// TIA Portal V19 export
FUNCTION_BLOCK "SmartLoopControl"   // FB182, LAD
TITLE = SMART LOOP CONTROLLER
// stored: Access Published, MemoryReserve 100, SetENOAutomatically false
   VAR_INPUT
      AreaInterfaceEntry : "AreaInterface";
      AreaInterfaceExit : "AreaInterface";
      DataIn : Struct
         Pb_StartStop : Bool;
         Pb_Start : Bool;
         Pb_Stop : Bool;
         SensorEntryMaterialPresence : Bool;
         SensorExitMaterialPresence : Bool;
         SensorExitEnableUseEncoder : Bool;
         SensorNotLoopMinHigh : Bool;   // FALSE = Min High
         SensorLoopMaxLow_Or_TPEntry : Bool;
         SensorLoopMaxLow_Or_TPExit : Bool;
         PlugConnected : Bool;
      END_STRUCT;
      CIn : "SmartLoopControl_CIn";
      Config : Struct
         PitTables_Exist : Bool := FALSE;
         Entry_PercentagePosError : LReal := 10.0;   // % Max Delta Counter position Vs Positions calculated from velocity
         Exit_PercentagePosError : LReal := 10.0;   // % Max Delta Counter position Vs Positions calculated from velocity
         Delay_CheckNoEntryBkwEnable : Time := T#6s;
         Delay_CheckNoEntryFwdEnable : Time := T#6s;
         Delay_CheckNoExitBkwEnable : Time := T#6s;
         Delay_CheckNoExitFwdEnable : Time := T#6s;
      END_STRUCT;
   END_VAR
   VAR_OUTPUT
      MachineInterfaceEntry : "MachineInterface";
      MachineInterfaceExit : "MachineInterface";
      COut : "SmartLoopControl_COut";
      DataOut : Struct
         LampSystemOn : Bool;
      END_STRUCT;
   END_VAR
   VAR_IN_OUT
      PersistentValues : Struct
         Par : "SmartLoopControl_Par";
      END_STRUCT;
   END_VAR
   VAR
      Ctrl : Struct
         RstAlarms : Bool;
         StopInPhase : Bool;
         StopProgrammed : Bool;
         StopAborting : Bool;
         ForceSyncFirstStart : Bool;
         ForceSyncMinHigh : Bool;
         ForceSyncCyclic : Bool;
         ForceSyncExt : Bool;
         ForceSync : Bool;
         Sync_Exe : Bool;
         Sync_EntryReduceOrStopFeed : Bool;
         Sync_ExitReduceOrStopFeed : Bool;
         MeasuringEnable : Bool;
         Entry_EnableFeedBkw : Bool;
         Entry_EnableFeedFwd : Bool;
         Exit_EnableFeedBkw : Bool;
         Exit_EnableFeedFwd : Bool;
         Entry_VelocityOverride : LReal;
         Exit_VelocityOverride : LReal;
         Exit_MaxAllowableFeedFwd : LReal;
      END_STRUCT;
      Sts : Struct
         IsStandstill : Bool;
         AlarmsPresence : Bool;
         WarningsPresence : Bool;
         SensorsMaxLow_OFF : Bool;
         SensorsMaxLow_ON : Bool;
         LoopMaterialCounterValid : Bool;
         SynchroRunning : Bool;
         CheckSensorCatchIsOn : Bool;
         CheckSensorLooseIsOn : Bool;
         WorkModeMatCounter : Bool;
         WorkModeSensors : Bool;
         SystemOn : Bool;
         MinHighReached : Bool;
         SynchroDone : Bool;
         CntFeedIncValid : Bool;
         AntiRepetitionForceSyncExt : Bool;
         Entry_MeasuringValuePosAxValid : Bool;
         Exit_MeasuringValuePosAxValid : Bool;
         Entry_MeasuringValueMatCounterValid : Bool;
         Exit_MeasuringValueMatCounterValid : Bool;
         SynchroDoneTof2s : Bool;
         MaxLowReached : Bool;
         SelectedPosStopMaxLow : LReal;
         SelectedOverrideScaling : LReal;
         LoopMaterialCounter : LReal;
         DifferenceInc : LReal;
         CntFeedIncPrevious : LReal;
         MissingToCyclicSync : LReal;
         SyncroMemLoopMaterialCounter : LReal;
         AntiRepetitionForceSyncExtSaveEntryMatCounter : LReal;
         AntiRepetitionForceSyncExtSaveExitMatCounter : LReal;
         EncEntry_MeasuringValuePosAx : LReal;
         EncExit_MeasuringValuePosAx : LReal;
         EncEntry_MeasuringValueMatCounter : LReal;
         EncExit_MeasuringValueMatCounter : LReal;
         LoopMaterialCounterOffset : LReal;
         LoopMaterialMissingToMaxLow : LReal;
         LoopMaterialMissingToMinHigh : LReal;
         Cases_Entry_VelocityOverride : UInt;
         Cases_Exit_VelocityOverride : UInt;
         Cases_Exit_MaxFeed : UInt;
         WorkMode : UInt;
      END_STRUCT;
      Wng : Struct
         NoAutReady : Bool;
         MeasInputsXORMeasuringValue : Bool;
         TimeOutCalculateLoopCounterOffset : Bool;
         SensorEnableEncIsOff : Bool;
         Entry_MatCounterNotValid : Bool;
         Exit_MatCounterNotValid : Bool;
         NotSystemOn : Bool;
         MinHighReached : Bool;
         SyncNeedToLooseSensor : Bool;
         SyncNeedToCatchSensor : Bool;
         Entry_NoBkwEnable : Bool;
         Entry_NoFwdEnable : Bool;
         Exit_NoBkwEnable : Bool;
         Exit_NoFwdEnable : Bool;
      END_STRUCT;
      Alr : Struct
         MeasInputsXORInputState : Bool;
         Entry_MatCounterLooseOfValidState : Bool;
         Exit_MatCounterLooseOfValidState : Bool;
         SensorError : Bool;
         PlugNotConnected : Bool;
         SyncSensorNotCatch : Bool;
         SyncSensorNotLoose : Bool;
         Entry_NoCounterMove : Bool;
         Exit_NoCounterMove : Bool;
      END_STRUCT;
      tonCheckMeasInputStateXOR : TON_TIME;
      tonDelaySensorMaxLowLoose { S7_SetPoint := 'True'} : TON_TIME;
      tonDelaySensorMaxLowCatch { S7_SetPoint := 'True'} : TON_TIME;
      tonCheckNoEntryCounterMove { S7_SetPoint := 'True'} : TON_TIME;
      tonCheckNoExitCounterMove { S7_SetPoint := 'True'} : TON_TIME;
      tonEnableForceSyncCyclic { S7_SetPoint := 'True'} : TON_TIME;
      tonSynchIdle { S7_SetPoint := 'True'} : TON_TIME;
      tonCheckBothMeasuringDone { S7_SetPoint := 'True'} : TON_TIME;
      tonTimeOutCalculateCounterOffset { S7_SetPoint := 'True'} : TON_TIME;
      tonSynchAutoReset { S7_SetPoint := 'True'} : TON_TIME;
      tof2sSynchroDone { S7_SetPoint := 'True'} : TON_TIME;
      tonRstMaterialCounterValid { S7_SetPoint := 'True'} : TON_TIME;
      tonSetMaxLow { S7_SetPoint := 'True'} : TON_TIME;
      tonRstMaxLow { S7_SetPoint := 'True'} : TON_TIME;
      tonCheckNoEntryBkwEnable { S7_SetPoint := 'True'} : TON_TIME;
      tonCheckNoEntryFwdEnable { S7_SetPoint := 'True'} : TON_TIME;
      tonCheckNoExitBkwEnable { S7_SetPoint := 'True'} : TON_TIME;
      tonCheckNoExitFwdEnable { S7_SetPoint := 'True'} : TON_TIME;
      SynchCycle { S7_SetPoint := 'True'} : UInt;
      CheckSensorCatchSaveLoopMaterialCounter : LReal;
      CheckSensorCatchFeeding : LReal;
      CheckSensorLooseSaveLoopMaterialCounter : LReal;
      CheckSensorLooseFeeding : LReal;
      AuxPbStartStopOneShot { S7_SetPoint := 'True'} : Bool;
      AuxSyncFirstStartOneShot : Bool;
      ModeMatCounterAndSystemOn : Bool;
      MinHighCumulative : Bool;
      AuxSyncMinHighOneShot : Bool;
      Entry_SaveMesInpID : UInt;
      Exit_SaveMesInpID : UInt;
      Check_Entry_Velocity { S7_SetPoint := 'True'} : "Check_Axis_Velocity";
      Check_Exit_Velocity { S7_SetPoint := 'True'} : "Check_Axis_Velocity";
   END_VAR
   VAR_TEMP
      PosMax : LReal;
      MaxMaterialInsideLoop : LReal;
      DeltaPosSync : LReal;
      DeltaPos : LReal;
      PbStartOneShot : Bool;
      PbStopOneShot : Bool;
      OK : Bool;
      Req : Bool;
      MinHighOverride : Bool;
      RstSynchro : Bool;
   END_VAR
   VAR CONSTANT
      DELTA_POS_LOOP_OVER_LOW_TABLE : LReal := 100.0;
      SYNCH_00_INIT : UInt := 0;
      SYNCH_01_ACTIVATE_MEASINPUTS : UInt := 1;
      SYNCH_10_IDLE : UInt := 10;
      SYNCH_11_CATCH_SENSOR : UInt := 11;
      SYNCH_12_LOOSE_SENSOR : UInt := 12;
      SYNCH_13_LAST_CATCH_SENSOR : UInt := 13;
      SYNCH_14_CALCULATE_COUNTER_OFFSET : UInt := 14;
      SYNCH_90_ERROR : UInt := 90;
      MODE_00_USE_SENSOR : UInt := 0;
      MODE_01_USE_MATERIAL_COUNTERS : UInt := 1;
      ENTRY_CASE_01_V0_ALARM_PRESENCE : UInt := 1;
      ENTRY_CASE_02_V0_MAX_LOW : UInt := 2;
      ENTRY_CASE_03_VMin_MAX_LOW_OVERRIDE : UInt := 3;
      ENTRY_CASE_04_V100_SYSTEM_OFF : UInt := 4;
      ENTRY_CASE_11_VMin_MODE_SENSORS : UInt := 11;
      ENTRY_CASE_12_VMax_MODE_SENSORS : UInt := 12;
      ENTRY_CASE_13_V100_MODE_SENSORS : UInt := 13;
      ENTRY_CASE_21_V100_SYNCHRO_RUNNING : UInt := 21;
      ENTRY_CASE_22_V0_SYNCHRO_RUNNING : UInt := 22;
      ENTRY_CASE_23_VMin_SYNCHRO_RUNNING : UInt := 23;
      ENTRY_CASE_24_VMin_MODE_COUNTERS : UInt := 24;
      ENTRY_CASE_25_VMed_MODE_COUNTERS : UInt := 25;
      ENTRY_CASE_26_VMax_MODE_COUNTERS : UInt := 26;
      ENTRY_CASE_27_VMaxMax_MODE_COUNTERS : UInt := 27;
      ENTRY_CASE_30_V100_UNKNOW : UInt := 30;
      EXIT_CASE_01_V0_ALARM_PRESENCE : UInt := 1;
      EXIT_CASE_02_0_MIN_HIGH : UInt := 2;
      EXIT_CASE_03_VMin_SYSTEM_OFF : UInt := 3;
      EXIT_CASE_04_VMin_NEXT_EMPTYING : UInt := 4;
      EXIT_CASE_05_VMax_EMPTYING : UInt := 5;
      EXIT_CASE_11_V100_MODE_SENSORS_OR_EXIT_MAN : UInt := 11;
      EXIT_CASE_12_VMIN_MODE_SENSORS_TEMPORARY : UInt := 12;
      EXIT_CASE_20_100_SYNCRO_RUNNING : UInt := 20;
      EXIT_CASE_21_0_SYNCRO_RUNNING : UInt := 21;
      EXIT_CASE_22_VMin_SYNCRO_RUNNING : UInt := 22;
      EXIT_CASE_23_VMin_MODE_COUNTERS : UInt := 23;
      EXIT_CASE_24_VMed_MODE_COUNTERS : UInt := 24;
      EXIT_CASE_25_VMax_MODE_COUNTERS : UInt := 25;
      EXIT_CASE_26_100_MODE_COUNTERS : UInt := 26;
      EXIT_MAX_FEED_CASE_1_NO_LIMIT : UInt := 1;
      EXIT_MAX_FEED_CASE_2_SYSTEM_OFF : UInt := 2;
      EXIT_MAX_FEED_CASE_3_NEXT_END_OF_MATERIAL : UInt := 3;
      EXIT_MAX_FEED_CASE_4_LOOP_MAT_COUNTER_NOT_VALID : UInt := 4;
      EXIT_MAX_FEED_CASE_5_LOOP_MAT_COUNTER_VALID : UInt := 5;
      EXIT_MAX_FEED_CASE_6_ALARM : UInt := 6;
      EXIT_MAX_FEED_CASE_7_MIN_HIGH_REACHED : UInt := 7;
   END_VAR
   VAR_TEMP   // added for the SCL form of the ladder/FBD networks
      _w1 : Bool;
      _w2 : Bool;
      _w3 : Bool;
      _w4 : Bool;
   END_VAR
BEGIN

REGION Network 1: Reset alarms
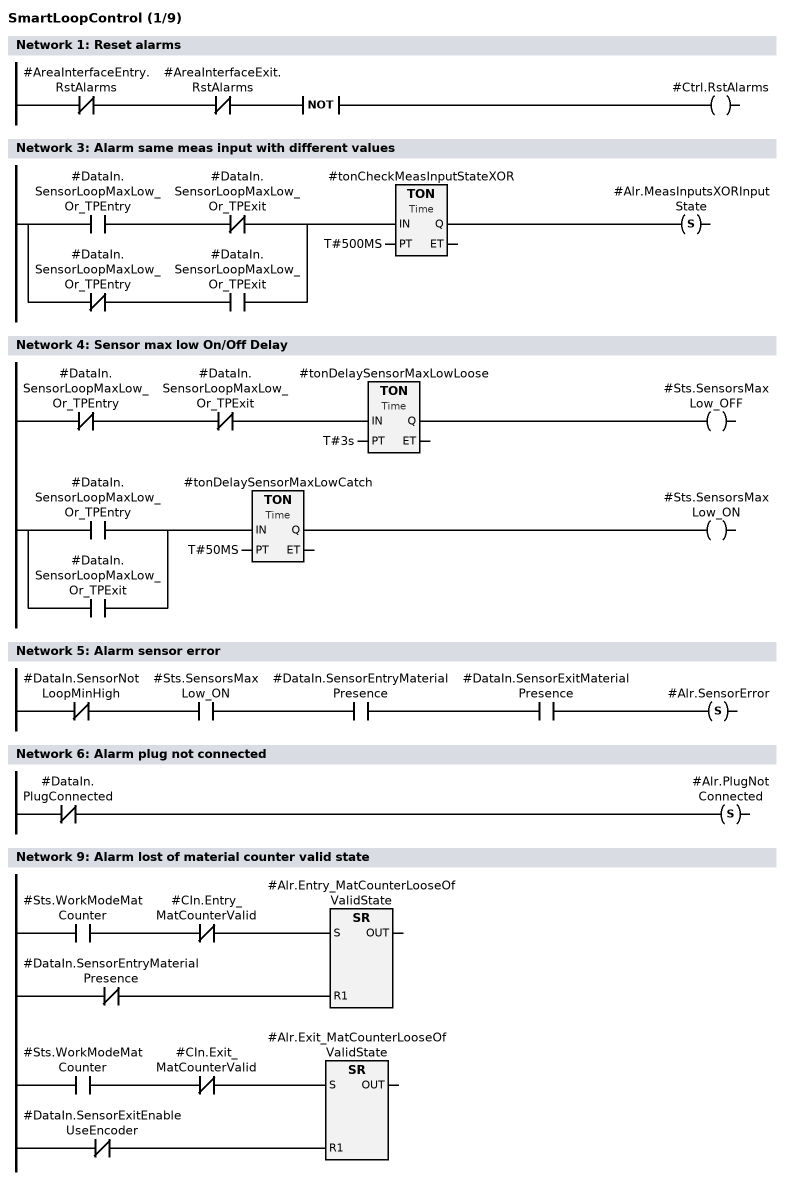
   RUNG wire#powerrail
      I_Contact( #AreaInterfaceEntry.RstAlarms )
      I_Contact( #AreaInterfaceExit.RstAlarms )
      Not()
      Coil( #Ctrl.RstAlarms )
   END_RUNG
   // the same network as SCL:
   #Ctrl.RstAlarms := NOT (NOT #AreaInterfaceEntry.RstAlarms AND NOT #AreaInterfaceExit.RstAlarms);
END_REGION

REGION Network 2 (SCL): Reset alarms execution
   IF #Ctrl.RstAlarms THEN
       #Wng.NoAutReady := FALSE;
       #Wng.MeasInputsXORMeasuringValue := FALSE;
       #Wng.TimeOutCalculateLoopCounterOffset := FALSE;
       #Wng.SensorEnableEncIsOff := FALSE;
       #Wng.Entry_MatCounterNotValid := FALSE;
       #Wng.Exit_MatCounterNotValid := FALSE;
       #Wng.NotSystemOn := FALSE;
       #Wng.MinHighReached := FALSE;
       #Wng.SyncNeedToLooseSensor := FALSE;
       #Wng.SyncNeedToCatchSensor := FALSE;
       #Wng.Entry_NoBkwEnable := FALSE;
       #Wng.Entry_NoFwdEnable := FALSE;
       #Wng.Exit_NoBkwEnable := FALSE;
       #Wng.Exit_NoFwdEnable := FALSE;

       #Alr.MeasInputsXORInputState := FALSE;
       #Alr.Entry_MatCounterLooseOfValidState := FALSE;
       #Alr.Exit_MatCounterLooseOfValidState := FALSE;
       #Alr.SensorError := FALSE;
       #Alr.SyncSensorNotCatch := FALSE;
       #Alr.SyncSensorNotLoose := FALSE;
       #Alr.Entry_NoCounterMove := FALSE;
       #Alr.Exit_NoCounterMove := FALSE;
       #Alr.PlugNotConnected := FALSE;

   END_IF;
END_REGION

REGION Network 3: Alarm same meas input with different values
   RUNG wire#powerrail
      Contact( #DataIn.SensorLoopMaxLow_Or_TPEntry )
      I_Contact( #DataIn.SensorLoopMaxLow_Or_TPExit )
      wire#w1
      { S7_Templates := "time_type := Time" } #tonCheckMeasInputStateXOR.TON(pt := T#500MS, et =>)
      S_Coil( #Alr.MeasInputsXORInputState )
   END_RUNG
   RUNG wire#powerrail
      I_Contact( #DataIn.SensorLoopMaxLow_Or_TPEntry )
      Contact( #DataIn.SensorLoopMaxLow_Or_TPExit )
   END_RUNG wire#w1
   // the same network as SCL:
   #tonCheckMeasInputStateXOR(IN := (#DataIn.SensorLoopMaxLow_Or_TPEntry AND NOT #DataIn.SensorLoopMaxLow_Or_TPExit) OR (NOT #DataIn.SensorLoopMaxLow_Or_TPEntry AND #DataIn.SensorLoopMaxLow_Or_TPExit),   // TON
                           PT := T#500MS);
   IF #tonCheckMeasInputStateXOR.Q THEN #Alr.MeasInputsXORInputState := TRUE; END_IF;
END_REGION

REGION Network 4: Sensor max low On/Off Delay
   RUNG wire#powerrail
      I_Contact( #DataIn.SensorLoopMaxLow_Or_TPEntry )
      I_Contact( #DataIn.SensorLoopMaxLow_Or_TPExit )
      { S7_Templates := "time_type := Time" } #tonDelaySensorMaxLowLoose.TON(pt := T#3s, et =>)
      Coil( #Sts.SensorsMaxLow_OFF )
   END_RUNG
   RUNG wire#powerrail
      Contact( #DataIn.SensorLoopMaxLow_Or_TPEntry )
      wire#w1
      { S7_Templates := "time_type := Time" } #tonDelaySensorMaxLowCatch.TON(pt := T#50MS, et =>)
      Coil( #Sts.SensorsMaxLow_ON )
   END_RUNG
   RUNG wire#powerrail
      Contact( #DataIn.SensorLoopMaxLow_Or_TPExit )
   END_RUNG wire#w1
   // the same network as SCL:
   #tonDelaySensorMaxLowLoose(IN := NOT #DataIn.SensorLoopMaxLow_Or_TPEntry AND NOT #DataIn.SensorLoopMaxLow_Or_TPExit,   // TON
                           PT := T#3s);
   #Sts.SensorsMaxLow_OFF := #tonDelaySensorMaxLowLoose.Q;
   #tonDelaySensorMaxLowCatch(IN := #DataIn.SensorLoopMaxLow_Or_TPEntry OR #DataIn.SensorLoopMaxLow_Or_TPExit,   // TON
                           PT := T#50MS);
   #Sts.SensorsMaxLow_ON := #tonDelaySensorMaxLowCatch.Q;
END_REGION

REGION Network 5: Alarm sensor error
   RUNG wire#powerrail
      I_Contact( #DataIn.SensorNotLoopMinHigh )
      Contact( #Sts.SensorsMaxLow_ON )
      Contact( #DataIn.SensorEntryMaterialPresence )
      Contact( #DataIn.SensorExitMaterialPresence )
      S_Coil( #Alr.SensorError )
   END_RUNG
   // the same network as SCL:
   IF NOT #DataIn.SensorNotLoopMinHigh AND #Sts.SensorsMaxLow_ON AND #DataIn.SensorEntryMaterialPresence AND #DataIn.SensorExitMaterialPresence THEN
       #Alr.SensorError := TRUE;
   END_IF;
END_REGION

REGION Network 6: Alarm plug not connected
   RUNG wire#powerrail
      I_Contact( #DataIn.PlugConnected )
      S_Coil( #Alr.PlugNotConnected )
   END_RUNG
   // the same network as SCL:
   IF NOT #DataIn.PlugConnected THEN #Alr.PlugNotConnected := TRUE; END_IF;
END_REGION

REGION Network 7 (SCL): Switch position Max Low / Middle as used Max Low
   IF  NOT #CIn.MaterialMiddlePos_Request
   THEN
       #Sts.SelectedPosStopMaxLow := #PersistentValues.Par.PosStopMaxLow;
       #Sts.SelectedOverrideScaling := 1.0;

   ELSE
       // Force value of middle position if is not properly setting
       IF NOT (#PersistentValues.Par.PosStopMiddle > #PersistentValues.Par.PosStopMinHigh
           AND
           #PersistentValues.Par.PosStopMiddle < #PersistentValues.Par.PosStopMaxLow)
       THEN
           #PersistentValues.Par.PosStopMiddle := #PersistentValues.Par.PosStopMinHigh + ((#PersistentValues.Par.PosStopMaxLow - #PersistentValues.Par.PosStopMinHigh) / 2.0);
       END_IF;

       // the new position for max low is the middle pistion
       #Sts.SelectedPosStopMaxLow := #PersistentValues.Par.PosStopMiddle;

       // this ratio is apply to all the position refered to max low (e.g. the limits for change exit velocity override)
       #Sts.SelectedOverrideScaling := #PersistentValues.Par.PosStopMiddle / #PersistentValues.Par.PosStopMaxLow;






   END_IF;
END_REGION

REGION Network 8 (SCL): Alarms Synch sensor (table) NOT catch / loose
   // !!! Se per qualche motivo il sensore di ansa bassa rimane sempre ON o sempre OFF c'è il rischio che durante il sincronismo dell'ansa no si verifichi mai l'evento di "sensore catturato" o "sensore perso" con conseguente riempimento eccessivo della
   // lamiera in ansa..Questi allami allarmi verificano se la quantità di lamiera rispetto al momento in cui è iniziato il controllo ha un valore coerente con la massima quantità possibile.
   #PosMax := MAX_LREAL(IN1 := #Sts.SelectedPosStopMaxLow, IN2 := #PersistentValues.Par.PosSynch);
   #MaxMaterialInsideLoop := #PosMax - #PersistentValues.Par.PosStopMinHigh;


   IF #Sts.LoopMaterialCounterValid AND #Sts.SynchroRunning THEN
       IF ((#SynchCycle = #SYNCH_11_CATCH_SENSOR) OR (#SynchCycle = #SYNCH_13_LAST_CATCH_SENSOR))
           AND NOT #Alr.SyncSensorNotCatch AND NOT #Sts.CheckSensorCatchIsOn
       THEN
           #Sts.CheckSensorCatchIsOn := TRUE;
           #CheckSensorCatchSaveLoopMaterialCounter := #Sts.LoopMaterialCounter;
       ELSIF ((#SynchCycle = #SYNCH_11_CATCH_SENSOR) OR (#SynchCycle = #SYNCH_13_LAST_CATCH_SENSOR))
           AND NOT #Alr.SyncSensorNotCatch AND #Sts.CheckSensorCatchIsOn
       THEN
           #CheckSensorCatchFeeding := ABS(#Sts.LoopMaterialCounter - #CheckSensorCatchSaveLoopMaterialCounter);
           IF #CheckSensorCatchFeeding > (1.5 * #MaxMaterialInsideLoop) THEN
               #Alr.SyncSensorNotCatch := TRUE;
           END_IF;
       ELSE
           #Sts.CheckSensorCatchIsOn := FALSE;
       END_IF;

       IF #SynchCycle = #SYNCH_12_LOOSE_SENSOR AND
           NOT #Alr.SyncSensorNotLoose AND NOT #Sts.CheckSensorLooseIsOn
       THEN
           #Sts.CheckSensorLooseIsOn := TRUE;
           #CheckSensorLooseSaveLoopMaterialCounter := #Sts.LoopMaterialCounter;
       ELSIF #SynchCycle = #SYNCH_12_LOOSE_SENSOR
           AND NOT #Alr.SyncSensorNotLoose AND #Sts.CheckSensorLooseIsOn
       THEN
           #CheckSensorLooseFeeding := ABS(#Sts.LoopMaterialCounter - #CheckSensorLooseSaveLoopMaterialCounter);
           IF #CheckSensorLooseFeeding > (1.5 * #MaxMaterialInsideLoop)
           THEN
               #Alr.SyncSensorNotLoose := TRUE;
           END_IF;
       ELSE
           #Sts.CheckSensorLooseIsOn := FALSE;
       END_IF;
   ELSE
       #Sts.CheckSensorCatchIsOn := FALSE;
       #Sts.CheckSensorLooseIsOn := FALSE;
   END_IF;
END_REGION

REGION Network 9: Alarm lost of material counter valid state
   RUNG wire#powerrail
      Contact( #Sts.WorkModeMatCounter )
      I_Contact( #CIn.Entry_MatCounterValid )
      S_SR(operand := #Alr.Entry_MatCounterLooseOfValidState, r1 := wire#w1)
   END_RUNG
   RUNG wire#powerrail
      I_Contact( #DataIn.SensorEntryMaterialPresence )
   END_RUNG wire#w1
   RUNG wire#powerrail
      Contact( #Sts.WorkModeMatCounter )
      I_Contact( #CIn.Exit_MatCounterValid )
      S_SR(operand := #Alr.Exit_MatCounterLooseOfValidState, r1 := wire#w2)
   END_RUNG
   RUNG wire#powerrail
      I_Contact( #DataIn.SensorExitEnableUseEncoder )
   END_RUNG wire#w2
   // the same network as SCL:
   IF #Sts.WorkModeMatCounter AND NOT #CIn.Entry_MatCounterValid THEN
       #Alr.Entry_MatCounterLooseOfValidState := TRUE;   // SR flip-flop
   END_IF;
   IF NOT #DataIn.SensorEntryMaterialPresence THEN #Alr.Entry_MatCounterLooseOfValidState := FALSE; END_IF;
   IF #Sts.WorkModeMatCounter AND NOT #CIn.Exit_MatCounterValid THEN
       #Alr.Exit_MatCounterLooseOfValidState := TRUE;   // SR flip-flop
   END_IF;
   IF NOT #DataIn.SensorExitEnableUseEncoder THEN #Alr.Exit_MatCounterLooseOfValidState := FALSE; END_IF;
END_REGION

REGION Network 10: Alarm no Entry counter move
   // sys.bypass = cambiare #Config.Entry_PercentagePosError in un 0/1 oppure valore time per il timer #tonCheckNoEntryCounterMove
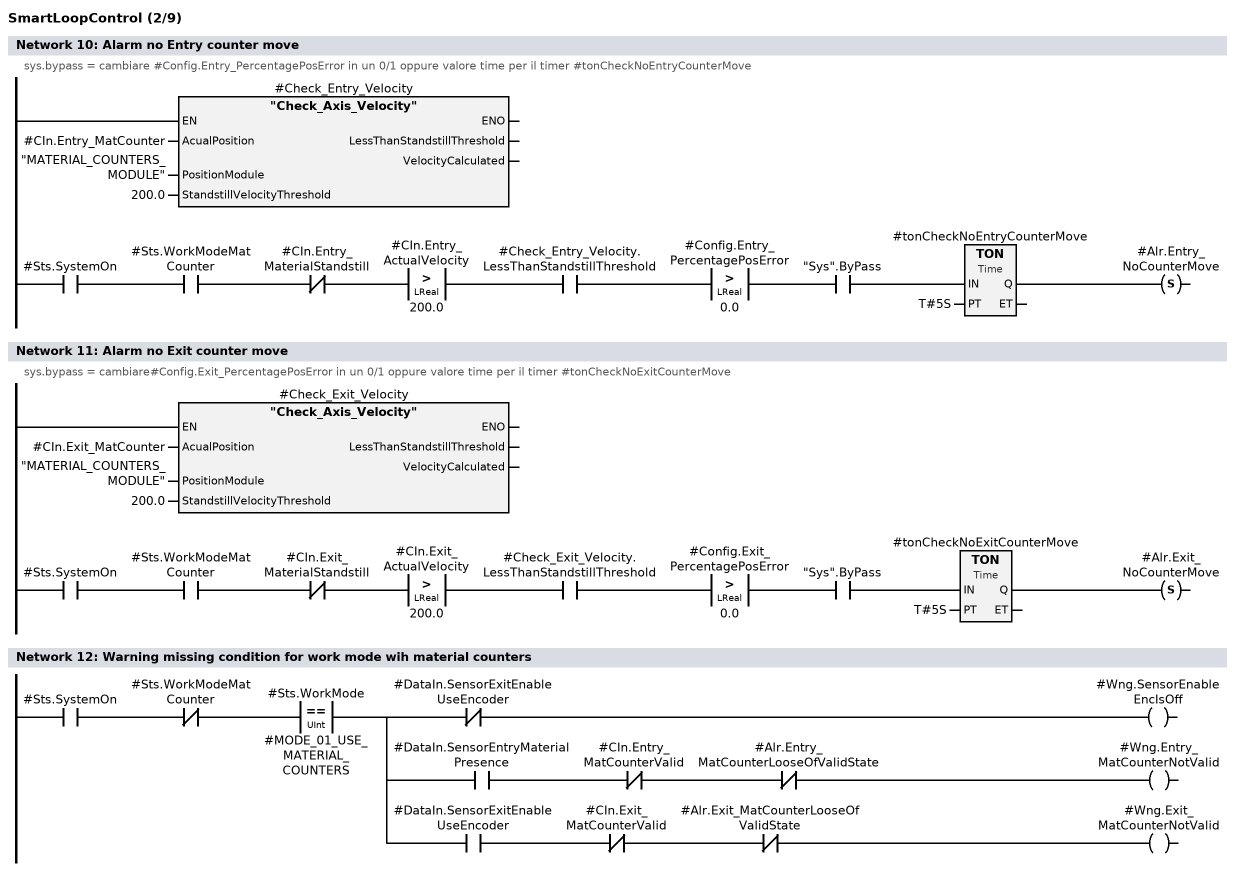
   RUNG wire#powerrail
      #Check_Entry_Velocity(AcualPosition := #CIn.Entry_MatCounter, PositionModule := "MATERIAL_COUNTERS_MODULE", StandstillVelocityThreshold := 200.0, LessThanStandstillThreshold =>, VelocityCalculated =>)
   END_RUNG
   RUNG wire#powerrail
      Contact( #Sts.SystemOn )
      Contact( #Sts.WorkModeMatCounter )
      I_Contact( #CIn.Entry_MaterialStandstill )
      { S7_Templates := "SrcType := LReal" } GT_Contact(in1 := #CIn.Entry_ActualVelocity, in2 := 200.0)
      Contact( #Check_Entry_Velocity.LessThanStandstillThreshold )
      { S7_Templates := "SrcType := LReal" } GT_Contact(in1 := #Config.Entry_PercentagePosError, in2 := 0.0)
      Contact( "Sys".ByPass )
      { S7_Templates := "time_type := Time" } #tonCheckNoEntryCounterMove.TON(pt := T#5S, et =>)
      S_Coil( #Alr.Entry_NoCounterMove )
   END_RUNG
   // the same network as SCL:
   #Check_Entry_Velocity(AcualPosition := #CIn.Entry_MatCounter,   // "Check_Axis_Velocity"
                         PositionModule := "MATERIAL_COUNTERS_MODULE",
                         StandstillVelocityThreshold := 200.0);
   #tonCheckNoEntryCounterMove(IN := #Sts.SystemOn AND #Sts.WorkModeMatCounter AND NOT #CIn.Entry_MaterialStandstill AND (#CIn.Entry_ActualVelocity > 200.0) AND #Check_Entry_Velocity.LessThanStandstillThreshold AND (#Config.Entry_PercentagePosError > 0.0) AND "Sys".ByPass,   // TON
                           PT := T#5S);
   IF #tonCheckNoEntryCounterMove.Q THEN #Alr.Entry_NoCounterMove := TRUE; END_IF;
END_REGION

REGION Network 11: Alarm no Exit counter move
   // sys.bypass = cambiare#Config.Exit_PercentagePosError in un 0/1 oppure valore time per il timer #tonCheckNoExitCounterMove
   RUNG wire#powerrail
      #Check_Exit_Velocity(AcualPosition := #CIn.Exit_MatCounter, PositionModule := "MATERIAL_COUNTERS_MODULE", StandstillVelocityThreshold := 200.0, LessThanStandstillThreshold =>, VelocityCalculated =>)
   END_RUNG
   RUNG wire#powerrail
      Contact( #Sts.SystemOn )
      Contact( #Sts.WorkModeMatCounter )
      I_Contact( #CIn.Exit_MaterialStandstill )
      { S7_Templates := "SrcType := LReal" } GT_Contact(in1 := #CIn.Exit_ActualVelocity, in2 := 200.0)
      Contact( #Check_Exit_Velocity.LessThanStandstillThreshold )
      { S7_Templates := "SrcType := LReal" } GT_Contact(in1 := #Config.Exit_PercentagePosError, in2 := 0.0)
      Contact( "Sys".ByPass )
      { S7_Templates := "time_type := Time" } #tonCheckNoExitCounterMove.TON(pt := T#5S, et =>)
      S_Coil( #Alr.Exit_NoCounterMove )
   END_RUNG
   // the same network as SCL:
   #Check_Exit_Velocity(AcualPosition := #CIn.Exit_MatCounter,   // "Check_Axis_Velocity"
                        PositionModule := "MATERIAL_COUNTERS_MODULE",
                        StandstillVelocityThreshold := 200.0);
   #tonCheckNoExitCounterMove(IN := #Sts.SystemOn AND #Sts.WorkModeMatCounter AND NOT #CIn.Exit_MaterialStandstill AND (#CIn.Exit_ActualVelocity > 200.0) AND #Check_Exit_Velocity.LessThanStandstillThreshold AND (#Config.Exit_PercentagePosError > 0.0) AND "Sys".ByPass,   // TON
                           PT := T#5S);
   IF #tonCheckNoExitCounterMove.Q THEN #Alr.Exit_NoCounterMove := TRUE; END_IF;
END_REGION

REGION Network 12: Warning missing condition for work mode wih material counters
   RUNG wire#powerrail
      Contact( #Sts.SystemOn )
      I_Contact( #Sts.WorkModeMatCounter )
      { S7_Templates := "SrcType := UInt" } EQ_Contact(in1 := #Sts.WorkMode, in2 := #MODE_01_USE_MATERIAL_COUNTERS)
      wire#w1
      I_Contact( #DataIn.SensorExitEnableUseEncoder )
      Coil( #Wng.SensorEnableEncIsOff )
   END_RUNG
   RUNG wire#w1
      Contact( #DataIn.SensorEntryMaterialPresence )
      I_Contact( #CIn.Entry_MatCounterValid )
      I_Contact( #Alr.Entry_MatCounterLooseOfValidState )
      Coil( #Wng.Entry_MatCounterNotValid )
   END_RUNG
   RUNG wire#w1
      Contact( #DataIn.SensorExitEnableUseEncoder )
      I_Contact( #CIn.Exit_MatCounterValid )
      I_Contact( #Alr.Exit_MatCounterLooseOfValidState )
      Coil( #Wng.Exit_MatCounterNotValid )
   END_RUNG
   // the same network as SCL:
   #_w1 := #Sts.SystemOn AND NOT #Sts.WorkModeMatCounter AND (#Sts.WorkMode = #MODE_01_USE_MATERIAL_COUNTERS);
   #Wng.SensorEnableEncIsOff := #_w1 AND NOT #DataIn.SensorExitEnableUseEncoder;
   #Wng.Entry_MatCounterNotValid := #_w1 AND #DataIn.SensorEntryMaterialPresence AND NOT #CIn.Entry_MatCounterValid AND NOT #Alr.Entry_MatCounterLooseOfValidState;
   #Wng.Exit_MatCounterNotValid := #_w1 AND #DataIn.SensorExitEnableUseEncoder AND NOT #CIn.Exit_MatCounterValid AND NOT #Alr.Exit_MatCounterLooseOfValidState;
END_REGION

REGION Network 13: Decoder working mode
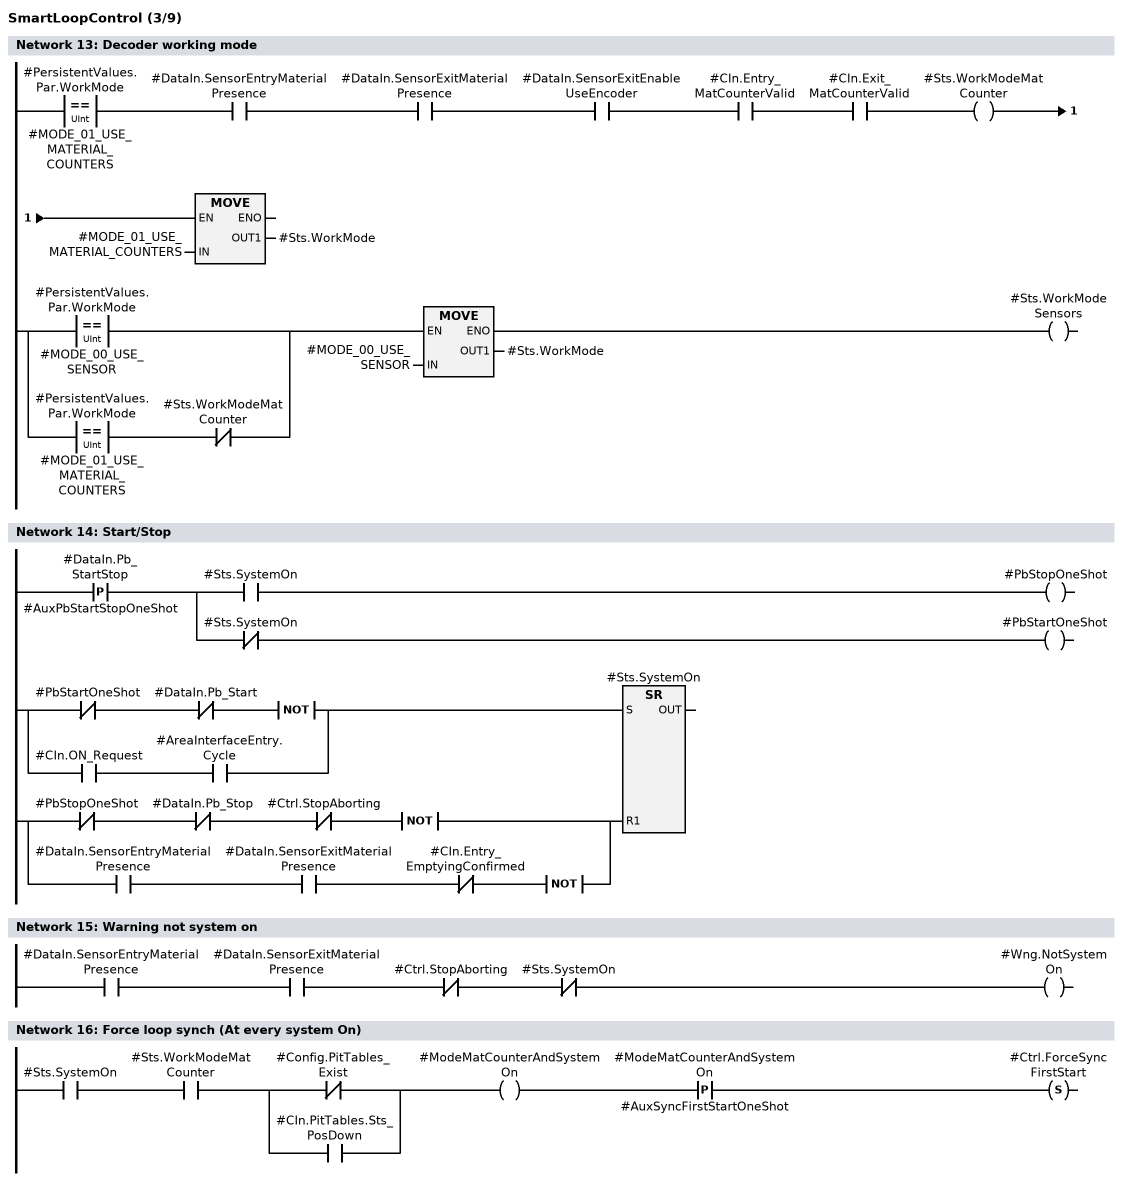
   RUNG wire#powerrail
      { S7_Templates := "SrcType := UInt" } EQ_Contact(in1 := #PersistentValues.Par.WorkMode, in2 := #MODE_01_USE_MATERIAL_COUNTERS)
      Contact( #DataIn.SensorEntryMaterialPresence )
      Contact( #DataIn.SensorExitMaterialPresence )
      Contact( #DataIn.SensorExitEnableUseEncoder )
      Contact( #CIn.Entry_MatCounterValid )
      Contact( #CIn.Exit_MatCounterValid )
      Coil( #Sts.WorkModeMatCounter )
      Move(in := #MODE_01_USE_MATERIAL_COUNTERS, out1 => #Sts.WorkMode)
   END_RUNG
   RUNG wire#powerrail
      { S7_Templates := "SrcType := UInt" } EQ_Contact(in1 := #PersistentValues.Par.WorkMode, in2 := #MODE_00_USE_SENSOR)
      wire#w1
      Move(in := #MODE_00_USE_SENSOR, out1 => #Sts.WorkMode)
      Coil( #Sts.WorkModeSensors )
   END_RUNG
   RUNG wire#powerrail
      { S7_Templates := "SrcType := UInt" } EQ_Contact(in1 := #PersistentValues.Par.WorkMode, in2 := #MODE_01_USE_MATERIAL_COUNTERS)
      I_Contact( #Sts.WorkModeMatCounter )
   END_RUNG wire#w1
   // the same network as SCL:
   #Sts.WorkModeMatCounter := (#PersistentValues.Par.WorkMode = #MODE_01_USE_MATERIAL_COUNTERS) AND #DataIn.SensorEntryMaterialPresence AND #DataIn.SensorExitMaterialPresence AND #DataIn.SensorExitEnableUseEncoder AND #CIn.Entry_MatCounterValid AND #CIn.Exit_MatCounterValid;
   IF #Sts.WorkModeMatCounter THEN #Sts.WorkMode := #MODE_01_USE_MATERIAL_COUNTERS; END_IF;
   #_w1 := (#PersistentValues.Par.WorkMode = #MODE_00_USE_SENSOR) OR ((#PersistentValues.Par.WorkMode = #MODE_01_USE_MATERIAL_COUNTERS) AND NOT #Sts.WorkModeMatCounter);
   IF #_w1 THEN #Sts.WorkMode := #MODE_00_USE_SENSOR; END_IF;
   #Sts.WorkModeSensors := #_w1;
END_REGION

REGION Network 14: Start/Stop
   RUNG wire#powerrail
      P_Contact(operand := #DataIn.Pb_StartStop, bit := #AuxPbStartStopOneShot)
      wire#w1
      Contact( #Sts.SystemOn )
      Coil( #PbStopOneShot )
   END_RUNG
   RUNG wire#w1
      I_Contact( #Sts.SystemOn )
      Coil( #PbStartOneShot )
   END_RUNG
   RUNG wire#powerrail
      I_Contact( #PbStartOneShot )
      I_Contact( #DataIn.Pb_Start )
      Not()
      wire#w2
      S_SR(operand := #Sts.SystemOn, r1 := wire#w3)
   END_RUNG
   RUNG wire#powerrail
      Contact( #CIn.ON_Request )
      Contact( #AreaInterfaceEntry.Cycle )
   END_RUNG wire#w2
   RUNG wire#powerrail
      I_Contact( #PbStopOneShot )
      I_Contact( #DataIn.Pb_Stop )
      I_Contact( #Ctrl.StopAborting )
      Not()
   END_RUNG wire#w3
   RUNG wire#powerrail
      Contact( #DataIn.SensorEntryMaterialPresence )
      Contact( #DataIn.SensorExitMaterialPresence )
      I_Contact( #CIn.Entry_EmptyingConfirmed )
      Not()
   END_RUNG wire#w3
   // the same network as SCL:
   #_w1 := #DataIn.Pb_StartStop AND NOT #AuxPbStartStopOneShot;   // rising edge of #DataIn.Pb_StartStop
   #AuxPbStartStopOneShot := #DataIn.Pb_StartStop;
   #PbStopOneShot := #_w1 AND #Sts.SystemOn;
   #PbStartOneShot := #_w1 AND NOT #Sts.SystemOn;
   IF NOT (NOT #PbStartOneShot AND NOT #DataIn.Pb_Start) OR (#CIn.ON_Request AND #AreaInterfaceEntry.Cycle) THEN
       #Sts.SystemOn := TRUE;   // SR flip-flop
   END_IF;
   IF NOT (NOT #PbStopOneShot AND NOT #DataIn.Pb_Stop AND NOT #Ctrl.StopAborting) OR NOT (#DataIn.SensorEntryMaterialPresence AND #DataIn.SensorExitMaterialPresence AND NOT #CIn.Entry_EmptyingConfirmed) THEN
       #Sts.SystemOn := FALSE;
   END_IF;
END_REGION

REGION Network 15: Warning not system on
   RUNG wire#powerrail
      Contact( #DataIn.SensorEntryMaterialPresence )
      Contact( #DataIn.SensorExitMaterialPresence )
      I_Contact( #Ctrl.StopAborting )
      I_Contact( #Sts.SystemOn )
      Coil( #Wng.NotSystemOn )
   END_RUNG
   // the same network as SCL:
   #Wng.NotSystemOn := #DataIn.SensorEntryMaterialPresence AND #DataIn.SensorExitMaterialPresence AND NOT #Ctrl.StopAborting AND NOT #Sts.SystemOn;
END_REGION

REGION Network 16: Force loop synch (At every system On)
   RUNG wire#powerrail
      Contact( #Sts.SystemOn )
      Contact( #Sts.WorkModeMatCounter )
      wire#w1
      I_Contact( #Config.PitTables_Exist )
      wire#w2
      Coil( #ModeMatCounterAndSystemOn )
      P_Contact(operand := #ModeMatCounterAndSystemOn, bit := #AuxSyncFirstStartOneShot)
      S_Coil( #Ctrl.ForceSyncFirstStart )
   END_RUNG
   RUNG wire#w1
      Contact( #CIn.PitTables.Sts_PosDown )
   END_RUNG wire#w2
   // the same network as SCL:
   #ModeMatCounterAndSystemOn := #Sts.SystemOn AND #Sts.WorkModeMatCounter AND (NOT #Config.PitTables_Exist OR #CIn.PitTables.Sts_PosDown);
   #_w1 := #ModeMatCounterAndSystemOn AND #ModeMatCounterAndSystemOn AND NOT #AuxSyncFirstStartOneShot;   // rising edge of #ModeMatCounterAndSystemOn
   #AuxSyncFirstStartOneShot := #ModeMatCounterAndSystemOn;
   IF #_w1 THEN #Ctrl.ForceSyncFirstStart := TRUE; END_IF;
END_REGION

REGION Network 17: Force loop synch each time min high sensor is engaged
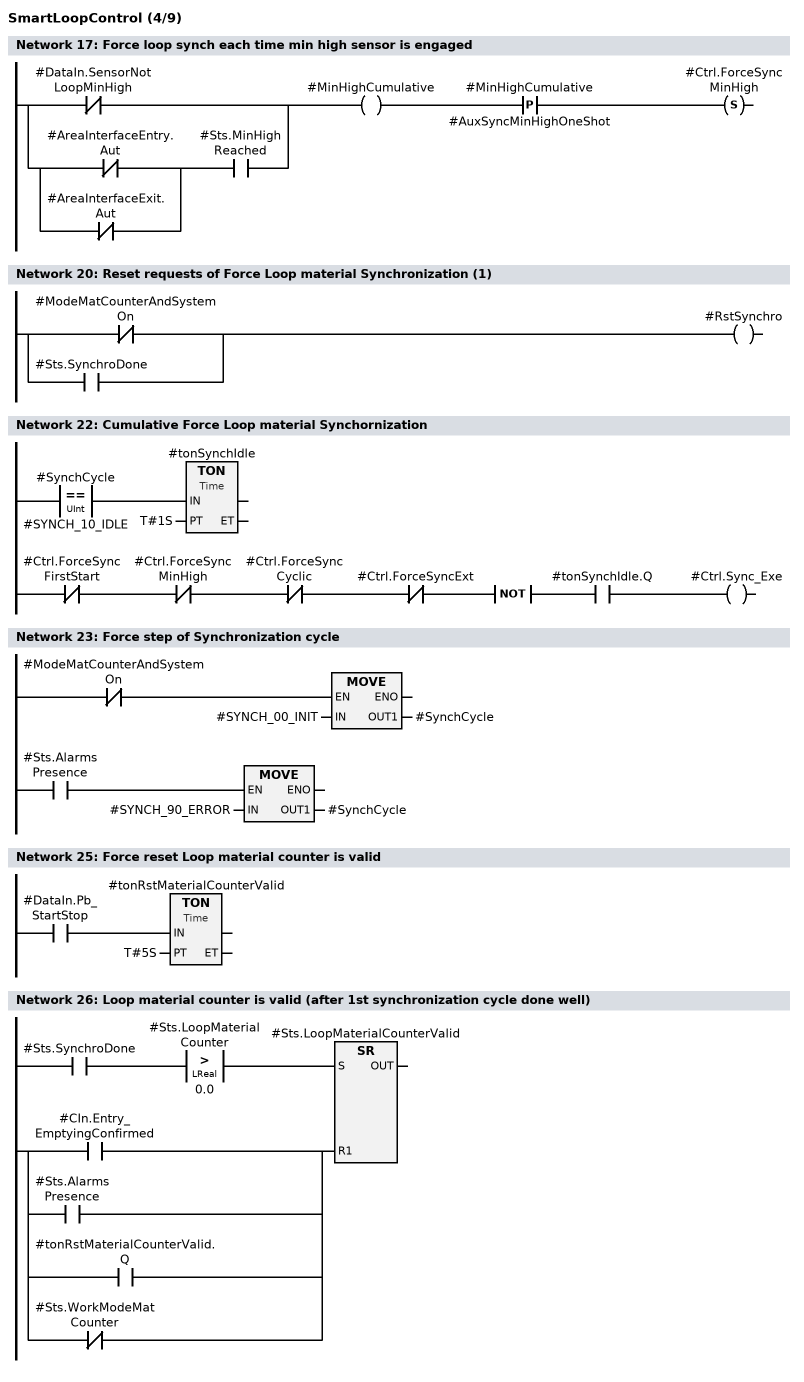
   RUNG wire#powerrail
      I_Contact( #DataIn.SensorNotLoopMinHigh )
      wire#w1
      Coil( #MinHighCumulative )
      P_Contact(operand := #MinHighCumulative, bit := #AuxSyncMinHighOneShot)
      S_Coil( #Ctrl.ForceSyncMinHigh )
   END_RUNG
   RUNG wire#powerrail
      I_Contact( #AreaInterfaceEntry.Aut )
      wire#w2
      Contact( #Sts.MinHighReached )
   END_RUNG wire#w1
   RUNG wire#powerrail
      I_Contact( #AreaInterfaceExit.Aut )
   END_RUNG wire#w2
   // the same network as SCL:
   #MinHighCumulative := NOT #DataIn.SensorNotLoopMinHigh OR ((NOT #AreaInterfaceEntry.Aut OR NOT #AreaInterfaceExit.Aut) AND #Sts.MinHighReached);
   #_w1 := #MinHighCumulative AND #MinHighCumulative AND NOT #AuxSyncMinHighOneShot;   // rising edge of #MinHighCumulative
   #AuxSyncMinHighOneShot := #MinHighCumulative;
   IF #_w1 THEN #Ctrl.ForceSyncMinHigh := TRUE; END_IF;
END_REGION

REGION Network 18 (SCL): Force Loop material Synchornization Cyclically
   #tonEnableForceSyncCyclic(IN:=NOT #Sts.SynchroDone AND NOT #Sts.SynchroRunning AND NOT #Ctrl.ForceSyncCyclic,PT:=T#1M);

   IF #Sts.SystemOn AND #Sts.WorkModeMatCounter AND #PersistentValues.Par.PosIntervalSynchroCyclic > 0.0 AND #tonEnableForceSyncCyclic.Q THEN

       // Detect increments of material loop Counter
       IF NOT #Sts.LoopMaterialCounterValid THEN
           #Sts.CntFeedIncValid := FALSE;
       ELSIF NOT #Sts.CntFeedIncValid THEN
           #Sts.CntFeedIncValid := TRUE;
           #Sts.DifferenceInc := 0.0;
           #Sts.CntFeedIncPrevious := #CIn.Exit_MatCounter;
       ELSIF #Sts.CntFeedIncValid THEN
           #Sts.DifferenceInc := "M_PosAMinusPosB"(PosA := #CIn.Exit_MatCounter, PosB := #Sts.CntFeedIncPrevious, MODULE := "MATERIAL_COUNTERS_MODULE");
           #Sts.CntFeedIncPrevious := #CIn.Exit_MatCounter;
           IF #Sts.DifferenceInc < 0.0 THEN
               #Sts.DifferenceInc := 0.0;
           END_IF;
       END_IF;

       // Filter of not possible increments
       IF #Sts.DifferenceInc > 0 AND #Sts.DifferenceInc <= 200.0 THEN
           #Sts.MissingToCyclicSync := #Sts.MissingToCyclicSync - #Sts.DifferenceInc;
       END_IF;

       // Trigger request
       IF (#Sts.MissingToCyclicSync < 0.0 OR #Sts.MissingToCyclicSync > #PersistentValues.Par.PosIntervalSynchroCyclic)
           AND NOT #CIn.Exit_MaterialStandstill AND NOT #CIn.Entry_MaterialStandstill
       THEN
           #Ctrl.ForceSyncCyclic := TRUE;
       END_IF;

   END_IF;
END_REGION

REGION Network 19 (SCL): Force Loop material Synchornization from external (e.g. tracking)
   IF #Sts.SynchroDone THEN

       #Sts.AntiRepetitionForceSyncExt := TRUE;
       #Sts.AntiRepetitionForceSyncExtSaveEntryMatCounter := #CIn.Entry_MatCounter;
       #Sts.AntiRepetitionForceSyncExtSaveExitMatCounter := #CIn.Exit_MatCounter;
       #Ctrl.ForceSyncExt := FALSE;

   ELSIF #Sts.AntiRepetitionForceSyncExt THEN

       IF #CIn.Entry_MatCounterValid THEN
           IF "M_CmpGT"(Xa := #CIn.Entry_MatCounter, Xb := "M_PosAPlusCostB"(PosA := #Sts.AntiRepetitionForceSyncExtSaveEntryMatCounter, CostB := #PersistentValues.Par.HysteresysSynchroExt, MODULE := "MATERIAL_COUNTERS_MODULE"), MODULE := "MATERIAL_COUNTERS_MODULE")
               AND
               "M_CmpGT"(Xa := #CIn.Exit_MatCounter, Xb := "M_PosAPlusCostB"(PosA := #Sts.AntiRepetitionForceSyncExtSaveExitMatCounter, CostB := #PersistentValues.Par.HysteresysSynchroExt, MODULE := "MATERIAL_COUNTERS_MODULE"), MODULE := "MATERIAL_COUNTERS_MODULE")
           THEN
               #Sts.AntiRepetitionForceSyncExt := FALSE;
           END_IF;
       ELSE
           #Sts.AntiRepetitionForceSyncExt := FALSE;
       END_IF;

   ELSIF #CIn.Synchro_Request AND NOT #Ctrl.ForceSyncExt THEN
       #Ctrl.ForceSyncExt := TRUE;
   END_IF;
END_REGION

REGION Network 20: Reset requests of Force Loop material Synchronization (1)
   RUNG wire#powerrail
      I_Contact( #ModeMatCounterAndSystemOn )
      wire#w1
      Coil( #RstSynchro )
   END_RUNG
   RUNG wire#powerrail
      Contact( #Sts.SynchroDone )
   END_RUNG wire#w1
   // the same network as SCL:
   #RstSynchro := NOT #ModeMatCounterAndSystemOn OR #Sts.SynchroDone;
END_REGION

REGION Network 21 (SCL): Reset requests of Force Loop material Synchronization (2)
   IF #RstSynchro THEN

       #Ctrl.ForceSyncFirstStart := FALSE;
       #Ctrl.ForceSyncMinHigh := FALSE;
       #Ctrl.ForceSyncCyclic := FALSE;
       #Ctrl.ForceSyncExt := FALSE;
       #Sts.SynchroDone := FALSE;
       #Sts.MissingToCyclicSync := #PersistentValues.Par.PosIntervalSynchroCyclic;

       IF #SynchCycle > 10 THEN
           #SynchCycle := 0;
       END_IF;


   END_IF;
END_REGION

REGION Network 22: Cumulative Force Loop material Synchornization
   RUNG wire#powerrail
      { S7_Templates := "SrcType := UInt" } EQ_Contact(in1 := #SynchCycle, in2 := #SYNCH_10_IDLE)
      { S7_Templates := "time_type := Time" } #tonSynchIdle.TON(pt := T#1S, et =>)
   END_RUNG
   RUNG wire#powerrail
      I_Contact( #Ctrl.ForceSyncFirstStart )
      I_Contact( #Ctrl.ForceSyncMinHigh )
      I_Contact( #Ctrl.ForceSyncCyclic )
      I_Contact( #Ctrl.ForceSyncExt )
      Not()
      Contact( #tonSynchIdle.Q )
      Coil( #Ctrl.Sync_Exe )
   END_RUNG
   // the same network as SCL:
   #tonSynchIdle(IN := #SynchCycle = #SYNCH_10_IDLE, PT := T#1S);   // TON
   #Ctrl.Sync_Exe := NOT (NOT #Ctrl.ForceSyncFirstStart AND NOT #Ctrl.ForceSyncMinHigh AND NOT #Ctrl.ForceSyncCyclic AND NOT #Ctrl.ForceSyncExt) AND #tonSynchIdle.Q;
END_REGION

REGION Network 23: Force step of Synchronization cycle
   RUNG wire#powerrail
      I_Contact( #ModeMatCounterAndSystemOn )
      Move(in := #SYNCH_00_INIT, out1 => #SynchCycle)
   END_RUNG
   RUNG wire#powerrail
      Contact( #Sts.AlarmsPresence )
      Move(in := #SYNCH_90_ERROR, out1 => #SynchCycle)
   END_RUNG
   // the same network as SCL:
   IF NOT #ModeMatCounterAndSystemOn THEN #SynchCycle := #SYNCH_00_INIT; END_IF;
   IF #Sts.AlarmsPresence THEN #SynchCycle := #SYNCH_90_ERROR; END_IF;
END_REGION

REGION Network 24 (SCL): Loop material Synchronization Cycle
   CASE #SynchCycle OF

       //-----------------------------------------------------------------------------------------------------------------
       // STATE 00 - INITIALIZATION
       //-----------------------------------------------------------------------------------------------------------------
       //
       #SYNCH_00_INIT:

           #Ctrl.Sync_EntryReduceOrStopFeed := FALSE;
           #Ctrl.Sync_ExitReduceOrStopFeed := FALSE;
           #Ctrl.MeasuringEnable := FALSE;

           IF #ModeMatCounterAndSystemOn
               (*
               AND NOT #CIn.Entry_MeasInput_InOperation
               AND NOT #CIn.Exit_MeasInput_InOperation
               *)
           THEN
               #SynchCycle := #SYNCH_01_ACTIVATE_MEASINPUTS;
           END_IF;

       //-----------------------------------------------------------------------------------------------------------------
       // STATE 01 - ACTIVATE MEASURING INPUTS
       //-----------------------------------------------------------------------------------------------------------------ù
       //
       #SYNCH_01_ACTIVATE_MEASINPUTS:

           #Ctrl.MeasuringEnable := TRUE;

           IF #CIn.Entry_MeasInput_InOperation AND #CIn.Exit_MeasInput_InOperation THEN
               #SynchCycle := #SYNCH_10_IDLE;

             //  #Entry_SaveMesInpID := #CIn.Entry_MeasInput_MeasuringDone_ID;
             //  #Exit_SaveMesInpID := #CIn.Exit_MeasInput_MeasuringDone_ID;
           END_IF;

       //-----------------------------------------------------------------------------------------------------------------
       // STATE 10 - WAIT SYNCHRO REQUEST
       //-----------------------------------------------------------------------------------------------------------------
       //
       #SYNCH_10_IDLE:

           #Ctrl.Sync_EntryReduceOrStopFeed := FALSE;
           #Ctrl.Sync_ExitReduceOrStopFeed := FALSE;

           #tonCheckBothMeasuringDone(IN := FALSE, PT := T#1S);
           #tonTimeOutCalculateCounterOffset(IN := FALSE, PT := T#5S);


           IF #Ctrl.Sync_Exe THEN

               #SynchCycle := #SYNCH_11_CATCH_SENSOR;

           END_IF;

       //-----------------------------------------------------------------------------------------------------------------
       // STATE 11 - CATCH TABLE SENSOR (MATERIAL DOWN) 
       //-----------------------------------------------------------------------------------------------------------------
       //
       #SYNCH_11_CATCH_SENSOR:

           #Ctrl.Sync_EntryReduceOrStopFeed := FALSE;
           #Ctrl.Sync_ExitReduceOrStopFeed := TRUE;

           IF #Sts.SensorsMaxLow_ON THEN

               #Sts.SyncroMemLoopMaterialCounter := #Sts.LoopMaterialCounter;


               #SynchCycle := #SYNCH_12_LOOSE_SENSOR;
           END_IF;

       //-----------------------------------------------------------------------------------------------------------------
       // STATE 12 - LOOSE TABLE SENSOR (MATERIAL UP) 
       //-----------------------------------------------------------------------------------------------------------------
       //
       #SYNCH_12_LOOSE_SENSOR:

           #Ctrl.Sync_EntryReduceOrStopFeed := TRUE;
           #Ctrl.Sync_ExitReduceOrStopFeed := FALSE;

           #tonCheckBothMeasuringDone(IN := FALSE, PT := T#1S);

           #DeltaPos :=  #Sts.SyncroMemLoopMaterialCounter - #Sts.LoopMaterialCounter;


           IF #Sts.SensorsMaxLow_OFF AND (#DeltaPos > #DELTA_POS_LOOP_OVER_LOW_TABLE) THEN

               #Entry_SaveMesInpID := #CIn.Entry_MeasInput_MeasuringDone_ID;
               #Exit_SaveMesInpID := #CIn.Exit_MeasInput_MeasuringDone_ID;

               #Ctrl.Sync_ExitReduceOrStopFeed := FALSE;
               #Sts.Entry_MeasuringValuePosAxValid := FALSE;
               #Sts.Exit_MeasuringValuePosAxValid := FALSE;
               #Sts.Entry_MeasuringValueMatCounterValid := FALSE;
               #Sts.Exit_MeasuringValueMatCounterValid := FALSE;

               #SynchCycle := #SYNCH_13_LAST_CATCH_SENSOR;

           END_IF;


       //-----------------------------------------------------------------------------------------------------------------
       // STATE 13 - LAST CATCH TABLE SENSOR (MATERIAL DOWN)
       //-----------------------------------------------------------------------------------------------------------------
       //
       #SYNCH_13_LAST_CATCH_SENSOR:

           #Ctrl.Sync_EntryReduceOrStopFeed := FALSE;
           #Ctrl.Sync_ExitReduceOrStopFeed := TRUE;

           #tonTimeOutCalculateCounterOffset(IN := FALSE, PT := T#5S);

           IF #CIn.Entry_MeasInput_MeasuringDone_ID <> #Entry_SaveMesInpID THEN
               #Sts.Entry_MeasuringValuePosAxValid := TRUE;
               #Sts.EncEntry_MeasuringValuePosAx := #CIn.Entry_MeasInput_MeasuringValue;

               #COut.Entry_AtSynch_PosAx := #Sts.EncEntry_MeasuringValuePosAx; // Valore in uscita per essere convertito in Pos.Mat.

           END_IF;

           IF #CIn.Exit_MeasInput_MeasuringDone_ID <> #Exit_SaveMesInpID THEN
               #Sts.Exit_MeasuringValuePosAxValid := TRUE;
               #Sts.EncExit_MeasuringValuePosAx := #CIn.Exit_MeasInput_MeasuringValue;

               #COut.Exit_AtSynch_PosAx := #Sts.EncExit_MeasuringValuePosAx; // Valore in uscita per essere convertito in Pos.Mat.
           END_IF;

           #OK := #Sts.Entry_MeasuringValuePosAxValid AND #Sts.Exit_MeasuringValuePosAxValid;

           #tonCheckBothMeasuringDone(IN := #Sts.SensorsMaxLow_ON AND NOT #OK,PT := T#1S);

           IF #Sts.SensorsMaxLow_ON AND #OK AND NOT #tonTimeOutCalculateCounterOffset.Q THEN

               #Ctrl.Sync_EntryReduceOrStopFeed := FALSE;
               #Ctrl.Sync_ExitReduceOrStopFeed := FALSE;
               #SynchCycle := #SYNCH_14_CALCULATE_COUNTER_OFFSET;

           ELSIF #tonCheckBothMeasuringDone.Q THEN
               #Wng.MeasInputsXORMeasuringValue := TRUE;
               #SynchCycle := #SYNCH_90_ERROR;
           END_IF;

       //-----------------------------------------------------------------------------------------------------------------
       // STATE 14 - CALCULATE LOOP COUNTER OFFSET
       //-----------------------------------------------------------------------------------------------------------------
       //
       #SYNCH_14_CALCULATE_COUNTER_OFFSET:

           #Ctrl.Sync_EntryReduceOrStopFeed := FALSE;
           #Ctrl.Sync_ExitReduceOrStopFeed := FALSE;

           #COut.Entry_AtSynch_PosAx := #Sts.EncEntry_MeasuringValuePosAx; // Valore in uscita per essere convertito in Pos.Mat.
           #COut.Exit_AtSynch_PosAx := #Sts.EncExit_MeasuringValuePosAx; // Valore in uscita per essere convertito in Pos.Mat.

           // Conversion encoder entry measured position form Pos.Ax to Pos.Material Counter
           IF #CIn.Entry_AtSinch_EchoPosAx = #COut.Entry_AtSynch_PosAx THEN
               #Sts.EncEntry_MeasuringValueMatCounter := #CIn.Entry_AtSynch_ConvertedPosMatCounter;
               #Sts.Entry_MeasuringValueMatCounterValid := TRUE;
           END_IF;

           // Conversion encoder exit measured position form Pos.Ax to Pos.Material Counter
           IF #CIn.Exit_AtSynch_ConvEchoPosAx = #COut.Exit_AtSynch_PosAx THEN
               #Sts.EncExit_MeasuringValueMatCounter := #CIn.Exit_AtSynch_ConvertedPosMatCounter;
               #Sts.Exit_MeasuringValueMatCounterValid := TRUE;
           END_IF;

           #tonTimeOutCalculateCounterOffset(IN := TRUE, PT := T#5S);

           IF #Sts.Entry_MeasuringValueMatCounterValid AND #Sts.Exit_MeasuringValueMatCounterValid THEN
               #DeltaPosSync := "M_PosAMinusPosB"(PosA := #Sts.EncEntry_MeasuringValueMatCounter, PosB := #Sts.EncExit_MeasuringValueMatCounter, MODULE := "MATERIAL_COUNTERS_MODULE");
               #Sts.LoopMaterialCounterOffset := #PersistentValues.Par.PosSynch - #DeltaPosSync;
               #Sts.SynchroDone := TRUE;
               #SynchCycle := #SYNCH_10_IDLE;

           ELSIF #tonTimeOutCalculateCounterOffset.Q THEN
               #Wng.TimeOutCalculateLoopCounterOffset := TRUE;
               #SynchCycle := #SYNCH_90_ERROR;
           END_IF;



       //----------------------------------------------
       // STATE 90 - SYNCH ERROR
       //----------------------------------------------
       //
       #SYNCH_90_ERROR:
           IF NOT #Sts.AlarmsPresence AND NOT #Wng.MeasInputsXORMeasuringValue AND NOT #Wng.TimeOutCalculateLoopCounterOffset THEN
               #SynchCycle := #SYNCH_00_INIT;
           END_IF;
   END_CASE;



   // Autoreset of synch cycle warnings
   #tonSynchAutoReset(IN:=#SynchCycle = #SYNCH_90_ERROR AND NOT #Alr.MeasInputsXORInputState ,PT:=T#3S);

   IF #tonSynchAutoReset.Q THEN
       #Wng.MeasInputsXORMeasuringValue := FALSE;
       #Wng.TimeOutCalculateLoopCounterOffset := FALSE;
   END_IF;

   #tof2sSynchroDone(IN:=#Sts.SynchroDone, PT:=T#2S);
   #Sts.SynchroDoneTof2s := #tof2sSynchroDone.Q;

   #Wng.SyncNeedToCatchSensor := #Ctrl.Sync_ExitReduceOrStopFeed;

   #Wng.SyncNeedToLooseSensor := #Ctrl.Sync_EntryReduceOrStopFeed;

   #Sts.SynchroRunning := (#SynchCycle > #SYNCH_10_IDLE) AND (#SynchCycle < #SYNCH_90_ERROR);
END_REGION

REGION Network 25: Force reset Loop material counter is valid
   RUNG wire#powerrail
      Contact( #DataIn.Pb_StartStop )
      { S7_Templates := "time_type := Time" } #tonRstMaterialCounterValid.TON(pt := T#5S, et =>)
   END_RUNG
   // the same network as SCL:
   #tonRstMaterialCounterValid(IN := #DataIn.Pb_StartStop, PT := T#5S);   // TON
END_REGION

REGION Network 26: Loop material counter is valid (after 1st synchronization cycle done well)
   RUNG wire#powerrail
      Contact( #Sts.SynchroDone )
      { S7_Templates := "SrcType := LReal" } GT_Contact(in1 := #Sts.LoopMaterialCounter, in2 := 0.0)
      S_SR(operand := #Sts.LoopMaterialCounterValid, r1 := wire#w1)
   END_RUNG
   RUNG wire#powerrail
      Contact( #CIn.Entry_EmptyingConfirmed )
   END_RUNG wire#w1
   RUNG wire#powerrail
      Contact( #Sts.AlarmsPresence )
   END_RUNG wire#w1
   RUNG wire#powerrail
      Contact( #tonRstMaterialCounterValid.Q )
   END_RUNG wire#w1
   RUNG wire#powerrail
      I_Contact( #Sts.WorkModeMatCounter )
   END_RUNG wire#w1
   // the same network as SCL:
   IF #Sts.SynchroDone AND (#Sts.LoopMaterialCounter > 0.0) THEN
       #Sts.LoopMaterialCounterValid := TRUE;   // SR flip-flop
   END_IF;
   IF #CIn.Entry_EmptyingConfirmed OR #Sts.AlarmsPresence OR #tonRstMaterialCounterValid.Q OR NOT #Sts.WorkModeMatCounter THEN
       #Sts.LoopMaterialCounterValid := FALSE;
   END_IF;
END_REGION

REGION Network 27 (SCL): Loop material counter
   // Material quantity inside loop
   #DeltaPos := "M_PosAMinusPosB"(PosA := #CIn.Entry_MatCounter, PosB := #CIn.Exit_MatCounter, MODULE := "MATERIAL_COUNTERS_MODULE");
   #Sts.LoopMaterialCounter := "M_PosAPlusCostB"(PosA := #DeltaPos, CostB := #Sts.LoopMaterialCounterOffset, MODULE := "MATERIAL_COUNTERS_MODULE");

   // Material missing to reach stop max low position
   #Sts.LoopMaterialMissingToMaxLow := "M_PosAMinusPosB"(PosA := #Sts.SelectedPosStopMaxLow, PosB := #Sts.LoopMaterialCounter, MODULE := "MATERIAL_COUNTERS_MODULE");

   // Material missing to reach stop min high position
   #Sts.LoopMaterialMissingToMinHigh := "M_PosAMinusPosB"(PosA := #Sts.LoopMaterialCounter, PosB := #PersistentValues.Par.PosStopMinHigh, MODULE := "MATERIAL_COUNTERS_MODULE");

   // Set to zero only for HMI visualization
   IF NOT #Sts.LoopMaterialCounterValid THEN
       #Sts.LoopMaterialMissingToMaxLow := 0.0;
       #Sts.LoopMaterialMissingToMinHigh := 0.0;
   END_IF;

   IF NOT #Sts.WorkModeMatCounter THEN
       #Sts.LoopMaterialCounter := 0.0;
   END_IF;
END_REGION

REGION Network 28 (SCL): Material Max Low Reached
   #tonSetMaxLow(IN:=#Sts.SensorsMaxLow_ON, PT:=#PersistentValues.Par.DlySetMaxLow);

   #tonRstMaxLow(IN:=#Sts.SensorsMaxLow_OFF, PT:=#PersistentValues.Par.DlyRstMaxLow);

   (*
   IF #CIn.Entry_MaxLowOverride THEN
       #Sts.MaxLowReached := FALSE;
     *)

   IF FALSE THEN
           ;

   ELSIF (#Sts.WorkModeSensors OR #Sts.SynchroRunning OR (#Sts.WorkModeMatCounter AND NOT #Sts.LoopMaterialCounterValid))
       AND
       (#tonSetMaxLow.Q OR (NOT #Sts.SystemOn AND #Sts.SensorsMaxLow_ON)) THEN
       #Sts.MaxLowReached := TRUE;

   ELSIF (#Sts.WorkModeSensors OR #Sts.SynchroRunning) AND (#tonRstMaxLow.Q OR (NOT #Sts.SystemOn AND #Sts.SensorsMaxLow_OFF)) THEN
       #Sts.MaxLowReached := FALSE;

   ELSIF #Sts.WorkModeMatCounter AND NOT #Sts.SynchroRunning AND #Sts.LoopMaterialCounterValid AND #Sts.LoopMaterialCounter > #Sts.SelectedPosStopMaxLow THEN
       #Sts.MaxLowReached := TRUE;

   ELSIF #Sts.WorkModeMatCounter AND #Sts.LoopMaterialCounter < (#Sts.SelectedPosStopMaxLow - (#PersistentValues.Par.PosDeltaRestartAfterMaxLow * #Sts.SelectedOverrideScaling)) THEN
       #Sts.MaxLowReached := FALSE;



   END_IF;
END_REGION

REGION Network 29: Bypass min high reached
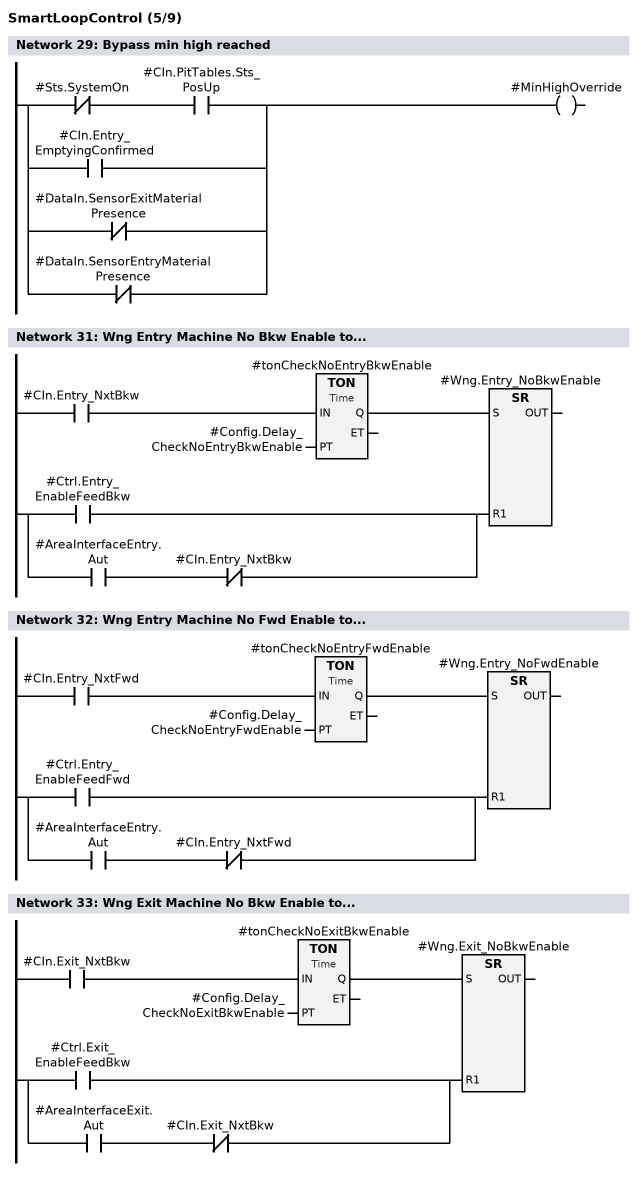
   RUNG wire#powerrail
      I_Contact( #Sts.SystemOn )
      Contact( #CIn.PitTables.Sts_PosUp )
      wire#w1
      Coil( #MinHighOverride )
   END_RUNG
   RUNG wire#powerrail
      Contact( #CIn.Entry_EmptyingConfirmed )
   END_RUNG wire#w1
   RUNG wire#powerrail
      I_Contact( #DataIn.SensorExitMaterialPresence )
   END_RUNG wire#w1
   RUNG wire#powerrail
      I_Contact( #DataIn.SensorEntryMaterialPresence )
   END_RUNG wire#w1
   // the same network as SCL:
   #MinHighOverride := (NOT #Sts.SystemOn AND #CIn.PitTables.Sts_PosUp) OR #CIn.Entry_EmptyingConfirmed OR NOT #DataIn.SensorExitMaterialPresence OR NOT #DataIn.SensorEntryMaterialPresence;
END_REGION

REGION Network 30 (SCL): Material Min High Reached
   IF #MinHighOverride THEN
       #Sts.MinHighReached := FALSE;

   ELSIF NOT #DataIn.SensorNotLoopMinHigh THEN
       #Sts.MinHighReached := TRUE;

   ELSIF NOT #Sts.SystemOn AND #AreaInterfaceExit.Man THEN
       #Sts.MinHighReached := FALSE;

   ELSIF #Sts.WorkModeSensors AND #Sts.SensorsMaxLow_ON THEN
       #Sts.MinHighReached := FALSE;


   ELSIF #Sts.WorkModeMatCounter AND #Sts.SynchroRunning THEN
       #Sts.MinHighReached := FALSE;

   ELSIF #Sts.WorkModeMatCounter AND #Sts.LoopMaterialCounterValid
       AND
       #Sts.LoopMaterialCounter <= #PersistentValues.Par.PosStopMinHigh THEN
       #Sts.MinHighReached := TRUE;

   ELSIF #Sts.WorkModeMatCounter AND #Sts.LoopMaterialCounterValid
       AND
       #Sts.LoopMaterialCounter > (#PersistentValues.Par.PosStopMinHigh + #PersistentValues.Par.PosDeltaRestartAfteMinHigh) THEN
       #Sts.MinHighReached := FALSE;

   ELSIF #Sts.WorkModeMatCounter AND #Sts.LoopMaterialCounterValid
       AND #Sts.MaxLowReached THEN
       #Sts.MinHighReached := FALSE;

   END_IF;

   #Wng.MinHighReached := #Sts.MinHighReached;
END_REGION

REGION Network 31: Wng Entry Machine No Bkw Enable to...
   RUNG wire#powerrail
      Contact( #CIn.Entry_NxtBkw )
      { S7_Templates := "time_type := Time" } #tonCheckNoEntryBkwEnable.TON(pt := #Config.Delay_CheckNoEntryBkwEnable, et =>)
      S_SR(operand := #Wng.Entry_NoBkwEnable, r1 := wire#w1)
   END_RUNG
   RUNG wire#powerrail
      Contact( #Ctrl.Entry_EnableFeedBkw )
   END_RUNG wire#w1
   RUNG wire#powerrail
      Contact( #AreaInterfaceEntry.Aut )
      I_Contact( #CIn.Entry_NxtBkw )
   END_RUNG wire#w1
   // the same network as SCL:
   #tonCheckNoEntryBkwEnable(IN := #CIn.Entry_NxtBkw, PT := #Config.Delay_CheckNoEntryBkwEnable);   // TON
   IF #tonCheckNoEntryBkwEnable.Q THEN
       #Wng.Entry_NoBkwEnable := TRUE;   // SR flip-flop
   END_IF;
   IF #Ctrl.Entry_EnableFeedBkw OR (#AreaInterfaceEntry.Aut AND NOT #CIn.Entry_NxtBkw) THEN
       #Wng.Entry_NoBkwEnable := FALSE;
   END_IF;
END_REGION

REGION Network 32: Wng Entry Machine No Fwd Enable to...
   RUNG wire#powerrail
      Contact( #CIn.Entry_NxtFwd )
      { S7_Templates := "time_type := Time" } #tonCheckNoEntryFwdEnable.TON(pt := #Config.Delay_CheckNoEntryFwdEnable, et =>)
      S_SR(operand := #Wng.Entry_NoFwdEnable, r1 := wire#w1)
   END_RUNG
   RUNG wire#powerrail
      Contact( #Ctrl.Entry_EnableFeedFwd )
   END_RUNG wire#w1
   RUNG wire#powerrail
      Contact( #AreaInterfaceEntry.Aut )
      I_Contact( #CIn.Entry_NxtFwd )
   END_RUNG wire#w1
   // the same network as SCL:
   #tonCheckNoEntryFwdEnable(IN := #CIn.Entry_NxtFwd, PT := #Config.Delay_CheckNoEntryFwdEnable);   // TON
   IF #tonCheckNoEntryFwdEnable.Q THEN
       #Wng.Entry_NoFwdEnable := TRUE;   // SR flip-flop
   END_IF;
   IF #Ctrl.Entry_EnableFeedFwd OR (#AreaInterfaceEntry.Aut AND NOT #CIn.Entry_NxtFwd) THEN
       #Wng.Entry_NoFwdEnable := FALSE;
   END_IF;
END_REGION

REGION Network 33: Wng Exit Machine No Bkw Enable to...
   RUNG wire#powerrail
      Contact( #CIn.Exit_NxtBkw )
      { S7_Templates := "time_type := Time" } #tonCheckNoExitBkwEnable.TON(pt := #Config.Delay_CheckNoExitBkwEnable, et =>)
      S_SR(operand := #Wng.Exit_NoBkwEnable, r1 := wire#w1)
   END_RUNG
   RUNG wire#powerrail
      Contact( #Ctrl.Exit_EnableFeedBkw )
   END_RUNG wire#w1
   RUNG wire#powerrail
      Contact( #AreaInterfaceExit.Aut )
      I_Contact( #CIn.Exit_NxtBkw )
   END_RUNG wire#w1
   // the same network as SCL:
   #tonCheckNoExitBkwEnable(IN := #CIn.Exit_NxtBkw, PT := #Config.Delay_CheckNoExitBkwEnable);   // TON
   IF #tonCheckNoExitBkwEnable.Q THEN
       #Wng.Exit_NoBkwEnable := TRUE;   // SR flip-flop
   END_IF;
   IF #Ctrl.Exit_EnableFeedBkw OR (#AreaInterfaceExit.Aut AND NOT #CIn.Exit_NxtBkw) THEN
       #Wng.Exit_NoBkwEnable := FALSE;
   END_IF;
END_REGION

REGION Network 34: Wng Exit Machine No Fwd Enable to...
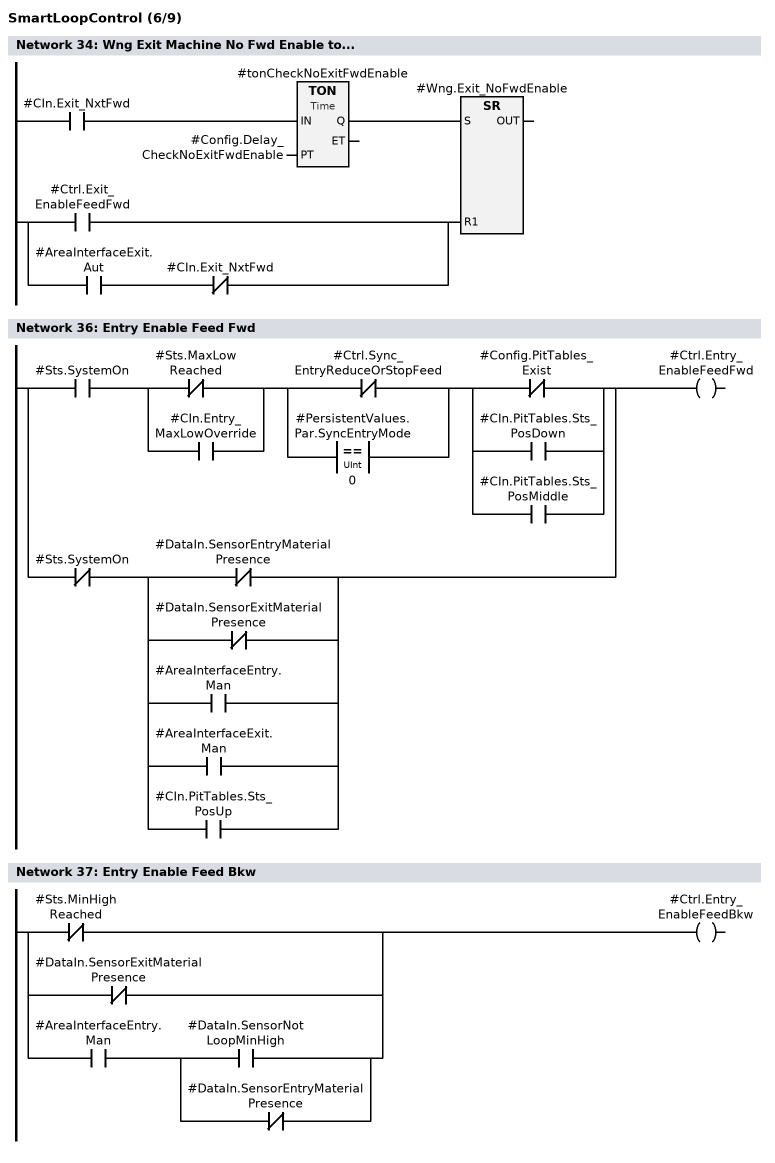
   RUNG wire#powerrail
      Contact( #CIn.Exit_NxtFwd )
      { S7_Templates := "time_type := Time" } #tonCheckNoExitFwdEnable.TON(pt := #Config.Delay_CheckNoExitFwdEnable, et =>)
      S_SR(operand := #Wng.Exit_NoFwdEnable, r1 := wire#w1)
   END_RUNG
   RUNG wire#powerrail
      Contact( #Ctrl.Exit_EnableFeedFwd )
   END_RUNG wire#w1
   RUNG wire#powerrail
      Contact( #AreaInterfaceExit.Aut )
      I_Contact( #CIn.Exit_NxtFwd )
   END_RUNG wire#w1
   // the same network as SCL:
   #tonCheckNoExitFwdEnable(IN := #CIn.Exit_NxtFwd, PT := #Config.Delay_CheckNoExitFwdEnable);   // TON
   IF #tonCheckNoExitFwdEnable.Q THEN
       #Wng.Exit_NoFwdEnable := TRUE;   // SR flip-flop
   END_IF;
   IF #Ctrl.Exit_EnableFeedFwd OR (#AreaInterfaceExit.Aut AND NOT #CIn.Exit_NxtFwd) THEN
       #Wng.Exit_NoFwdEnable := FALSE;
   END_IF;
END_REGION

REGION Network 35 (SCL): Cycle stop
   // Cycle Stop in phase
   IF NOT #AreaInterfaceEntry.StopInPhase AND NOT #AreaInterfaceExit.StopInPhase THEN
       #Ctrl.StopInPhase := FALSE;
   ELSIF #CIn.EnableStopInPhase THEN
       #Ctrl.StopInPhase := TRUE;
   END_IF;

   // Cycle Stop programmed
   IF NOT #AreaInterfaceEntry.StopProgrammed AND NOT #AreaInterfaceExit.StopProgrammed THEN
       #Ctrl.StopProgrammed := FALSE;
   ELSIF #CIn.EnableStopProgrammed THEN
       #Ctrl.StopProgrammed := TRUE;
   END_IF;
END_REGION

REGION Network 36: Entry Enable Feed Fwd
   RUNG wire#powerrail
      Contact( #Sts.SystemOn )
      wire#w1
      I_Contact( #Sts.MaxLowReached )
      wire#w2
      I_Contact( #Ctrl.Sync_EntryReduceOrStopFeed )
      wire#w3
      I_Contact( #Config.PitTables_Exist )
      wire#w4
      Coil( #Ctrl.Entry_EnableFeedFwd )
   END_RUNG
   RUNG wire#w1
      Contact( #CIn.Entry_MaxLowOverride )
   END_RUNG wire#w2
   RUNG wire#w2
      { S7_Templates := "SrcType := UInt" } EQ_Contact(in1 := #PersistentValues.Par.SyncEntryMode, in2 := 0)
   END_RUNG wire#w3
   RUNG wire#w3
      Contact( #CIn.PitTables.Sts_PosDown )
   END_RUNG wire#w4
   RUNG wire#w3
      Contact( #CIn.PitTables.Sts_PosMiddle )
   END_RUNG wire#w4
   RUNG wire#powerrail
      I_Contact( #Sts.SystemOn )
      wire#w5
      I_Contact( #DataIn.SensorEntryMaterialPresence )
   END_RUNG wire#w4
   RUNG wire#w5
      I_Contact( #DataIn.SensorExitMaterialPresence )
   END_RUNG wire#w4
   RUNG wire#w5
      Contact( #AreaInterfaceEntry.Man )
   END_RUNG wire#w4
   RUNG wire#w5
      Contact( #AreaInterfaceExit.Man )
   END_RUNG wire#w4
   RUNG wire#w5
      Contact( #CIn.PitTables.Sts_PosUp )
   END_RUNG wire#w4
   // the same network as SCL:
   #Ctrl.Entry_EnableFeedFwd := (#Sts.SystemOn AND (NOT #Sts.MaxLowReached OR #CIn.Entry_MaxLowOverride) AND (NOT #Ctrl.Sync_EntryReduceOrStopFeed OR (#PersistentValues.Par.SyncEntryMode = 0)) AND (NOT #Config.PitTables_Exist OR #CIn.PitTables.Sts_PosDown OR #CIn.PitTables.Sts_PosMiddle)) OR (NOT #Sts.SystemOn AND (NOT #DataIn.SensorEntryMaterialPresence OR NOT #DataIn.SensorExitMaterialPresence OR #AreaInterfaceEntry.Man OR #AreaInterfaceExit.Man OR #CIn.PitTables.Sts_PosUp));
END_REGION

REGION Network 37: Entry Enable Feed Bkw
   RUNG wire#powerrail
      I_Contact( #Sts.MinHighReached )
      wire#w1
      Coil( #Ctrl.Entry_EnableFeedBkw )
   END_RUNG
   RUNG wire#powerrail
      I_Contact( #DataIn.SensorExitMaterialPresence )
   END_RUNG wire#w1
   RUNG wire#powerrail
      Contact( #AreaInterfaceEntry.Man )
      wire#w2
      Contact( #DataIn.SensorNotLoopMinHigh )
   END_RUNG wire#w1
   RUNG wire#w2
      I_Contact( #DataIn.SensorEntryMaterialPresence )
   END_RUNG wire#w1
   // the same network as SCL:
   #Ctrl.Entry_EnableFeedBkw := NOT #Sts.MinHighReached OR NOT #DataIn.SensorExitMaterialPresence OR (#AreaInterfaceEntry.Man AND (#DataIn.SensorNotLoopMinHigh OR NOT #DataIn.SensorEntryMaterialPresence));
END_REGION

REGION Network 38: Exit machine enable feed forward
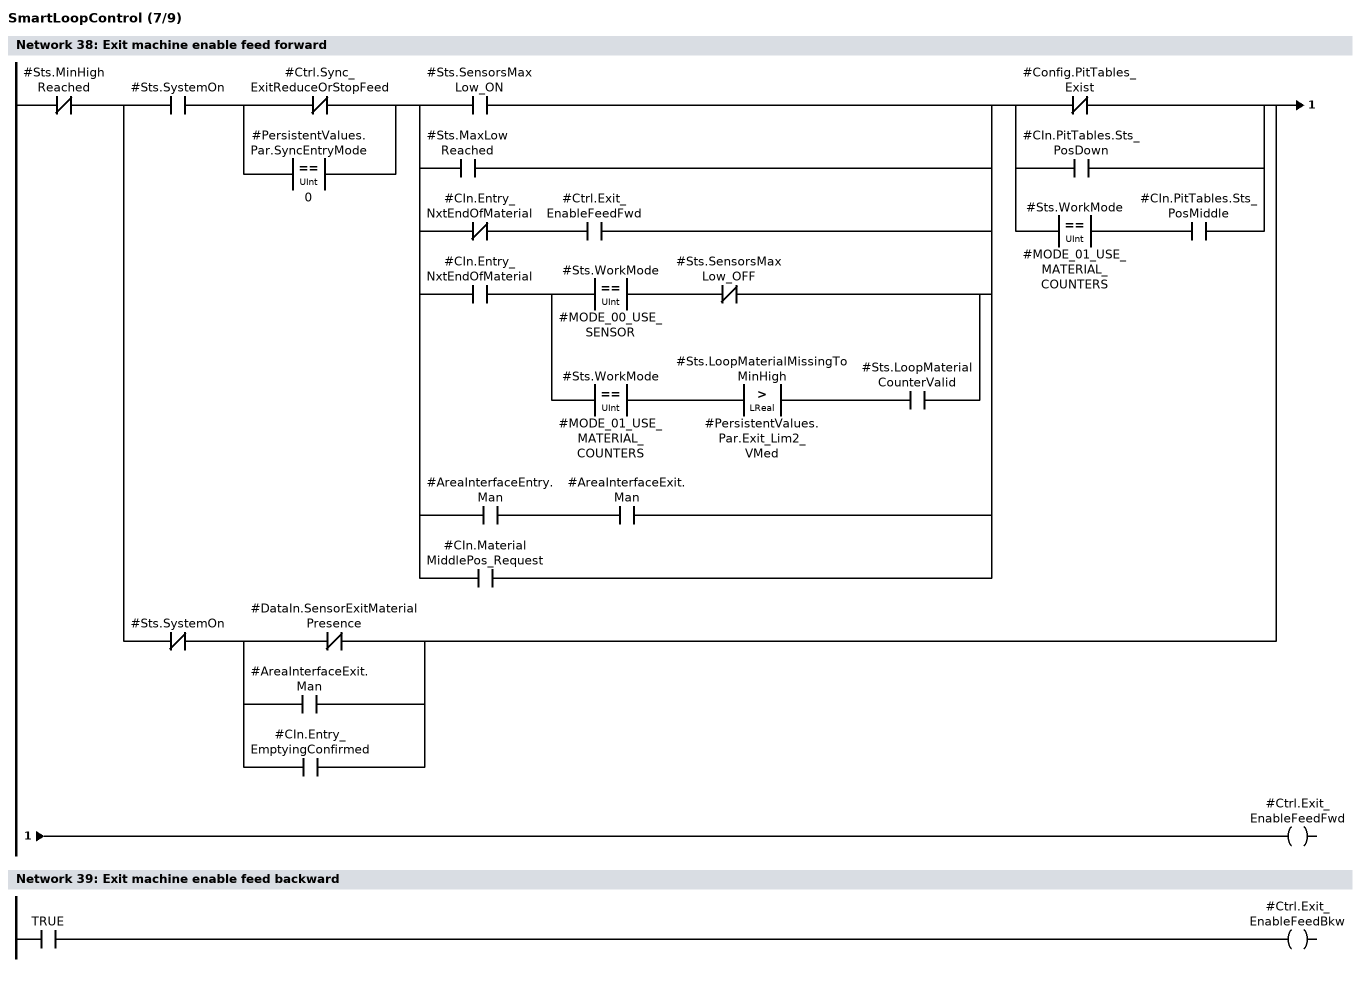
   RUNG wire#powerrail
      I_Contact( #Sts.MinHighReached )
      wire#w1
      Contact( #Sts.SystemOn )
      wire#w2
      I_Contact( #Ctrl.Sync_ExitReduceOrStopFeed )
      wire#w3
      Contact( #Sts.SensorsMaxLow_ON )
      wire#w4
      I_Contact( #Config.PitTables_Exist )
      wire#w6
      Coil( #Ctrl.Exit_EnableFeedFwd )
   END_RUNG
   RUNG wire#w2
      { S7_Templates := "SrcType := UInt" } EQ_Contact(in1 := #PersistentValues.Par.SyncEntryMode, in2 := 0)
   END_RUNG wire#w3
   RUNG wire#w3
      Contact( #Sts.MaxLowReached )
   END_RUNG wire#w4
   RUNG wire#w3
      I_Contact( #CIn.Entry_NxtEndOfMaterial )
      Contact( #Ctrl.Exit_EnableFeedFwd )
   END_RUNG wire#w4
   RUNG wire#w3
      Contact( #CIn.Entry_NxtEndOfMaterial )
      wire#w5
      { S7_Templates := "SrcType := UInt" } EQ_Contact(in1 := #Sts.WorkMode, in2 := #MODE_00_USE_SENSOR)
      I_Contact( #Sts.SensorsMaxLow_OFF )
   END_RUNG wire#w4
   RUNG wire#w5
      { S7_Templates := "SrcType := UInt" } EQ_Contact(in1 := #Sts.WorkMode, in2 := #MODE_01_USE_MATERIAL_COUNTERS)
      { S7_Templates := "SrcType := LReal" } GT_Contact(in1 := #Sts.LoopMaterialMissingToMinHigh, in2 := #PersistentValues.Par.Exit_Lim2_VMed)
      Contact( #Sts.LoopMaterialCounterValid )
   END_RUNG wire#w4
   RUNG wire#w3
      Contact( #AreaInterfaceEntry.Man )
      Contact( #AreaInterfaceExit.Man )
   END_RUNG wire#w4
   RUNG wire#w3
      Contact( #CIn.MaterialMiddlePos_Request )
   END_RUNG wire#w4
   RUNG wire#w4
      Contact( #CIn.PitTables.Sts_PosDown )
   END_RUNG wire#w6
   RUNG wire#w4
      { S7_Templates := "SrcType := UInt" } EQ_Contact(in1 := #Sts.WorkMode, in2 := #MODE_01_USE_MATERIAL_COUNTERS)
      Contact( #CIn.PitTables.Sts_PosMiddle )
   END_RUNG wire#w6
   RUNG wire#w1
      I_Contact( #Sts.SystemOn )
      wire#w7
      I_Contact( #DataIn.SensorExitMaterialPresence )
   END_RUNG wire#w6
   RUNG wire#w7
      Contact( #AreaInterfaceExit.Man )
   END_RUNG wire#w6
   RUNG wire#w7
      Contact( #CIn.Entry_EmptyingConfirmed )
   END_RUNG wire#w6
   // the same network as SCL:
   #Ctrl.Exit_EnableFeedFwd := NOT #Sts.MinHighReached AND ((#Sts.SystemOn AND (NOT #Ctrl.Sync_ExitReduceOrStopFeed OR (#PersistentValues.Par.SyncEntryMode = 0)) AND (#Sts.SensorsMaxLow_ON OR #Sts.MaxLowReached OR (NOT #CIn.Entry_NxtEndOfMaterial AND #Ctrl.Exit_EnableFeedFwd) OR (#CIn.Entry_NxtEndOfMaterial AND (((#Sts.WorkMode = #MODE_00_USE_SENSOR) AND NOT #Sts.SensorsMaxLow_OFF) OR ((#Sts.WorkMode = #MODE_01_USE_MATERIAL_COUNTERS) AND (#Sts.LoopMaterialMissingToMinHigh > #PersistentValues.Par.Exit_Lim2_VMed) AND #Sts.LoopMaterialCounterValid))) OR (#AreaInterfaceEntry.Man AND #AreaInterfaceExit.Man) OR #CIn.MaterialMiddlePos_Request) AND (NOT #Config.PitTables_Exist OR #CIn.PitTables.Sts_PosDown OR ((#Sts.WorkMode = #MODE_01_USE_MATERIAL_COUNTERS) AND #CIn.PitTables.Sts_PosMiddle))) OR (NOT #Sts.SystemOn AND (NOT #DataIn.SensorExitMaterialPresence OR #AreaInterfaceExit.Man OR #CIn.Entry_EmptyingConfirmed)));
END_REGION

REGION Network 39: Exit machine enable feed backward
   RUNG wire#powerrail
      Contact( TRUE )
      Coil( #Ctrl.Exit_EnableFeedBkw )
   END_RUNG
   // the same network as SCL:
   #Ctrl.Exit_EnableFeedBkw := TRUE;
END_REGION

REGION Network 40 (SCL): Entry Velocity override
   //=================================================================================================     
   // Entry machine velocity override
   //=================================================================================================     

   // CASE 01 -> 0% when alarm presence
   // 
   IF #Sts.AlarmsPresence THEN
       #Ctrl.Entry_VelocityOverride := 0.0;
       #Sts.Cases_Entry_VelocityOverride := #ENTRY_CASE_01_V0_ALARM_PRESENCE;


   // CASE 02 -> 0% if Max Low reached and not Max low override 
   // 
   ELSIF #Sts.MaxLowReached AND NOT #CIn.Entry_MaxLowOverride  THEN
       #Ctrl.Entry_VelocityOverride := 0.0;

       IF NOT #tonSetMaxLow.Q THEN
           #Ctrl.Entry_VelocityOverride := 0.1;
       END_IF;
       #Sts.Cases_Entry_VelocityOverride := #ENTRY_CASE_02_V0_MAX_LOW;


   // CASE 03 -> VMin when max low overriden and system ON
   // 
   ELSIF #CIn.Entry_MaxLowOverride AND #Sts.SystemOn THEN

       #Ctrl.Entry_VelocityOverride := #PersistentValues.Par.Entry_Override1_VMin;

       #Sts.Cases_Entry_VelocityOverride := #ENTRY_CASE_03_VMin_MAX_LOW_OVERRIDE;

   // CASE 04 -> 100% when system is off
   // 
   ELSIF NOT #Sts.SystemOn THEN
       #Ctrl.Entry_VelocityOverride := 100.0;
       #Sts.Cases_Entry_VelocityOverride := #ENTRY_CASE_04_V100_SYSTEM_OFF;



   //°°°°°°°°°°°°°°°°°°°°°°°°°°°°°°°°°°°°°°°°°°°°°°°°°°°°°°°°°°°°°°°°°°°°°°°°°°°°°°°°°°°°°°°°°°°°°°°°°°°°°°°°°°°°°
   // CASES 11..13 When working mode = Sensors
   //°°°°°°°°°°°°°°°°°°°°°°°°°°°°°°°°°°°°°°°°°°°°°°°°°°°°°°°°°°°°°°°°°°°°°°°°°°°°°°°°°°°°°°°°°°°°°°°°°°°°°°°°°°°°°
   //
   ELSIF #Sts.WorkModeSensors THEN
       // CASE 11 -> working mode = Sensors; VMin if table sensor is engagged but time for stop is not elapsed
       IF #Sts.SensorsMaxLow_ON THEN
           #Ctrl.Entry_VelocityOverride := #PersistentValues.Par.Entry_Override1_VMin;
           #Sts.Cases_Entry_VelocityOverride := #ENTRY_CASE_11_VMin_MODE_SENSORS;
           // CASE 12 -> working mode = Sensors; VMax if not Min High Reached
       ELSIF NOT #Sts.MinHighReached THEN
           #Ctrl.Entry_VelocityOverride := #PersistentValues.Par.Entry_Override3_VMax;
           #Sts.Cases_Entry_VelocityOverride := #ENTRY_CASE_12_VMax_MODE_SENSORS;
           // CASE 13 -> working mode = Sensors; 100% Min High Reached
       ELSIF #Sts.MinHighReached THEN
           #Ctrl.Entry_VelocityOverride := 100.0;
           #Sts.Cases_Entry_VelocityOverride := #ENTRY_CASE_13_V100_MODE_SENSORS;
       END_IF;

   //
   // 
   //°°°°°°°°°°°°°°°°°°°°°°°°°°°°°°°°°°°°°°°°°°°°°°°°°°°°°°°°°°°°°°°°°°°°°°°°°°°°°°°°°°°°°°°°°°°°°°°°°°°°°°°°°°°°°
   // CASES 21..26 When working mode = Material Counters
   //°°°°°°°°°°°°°°°°°°°°°°°°°°°°°°°°°°°°°°°°°°°°°°°°°°°°°°°°°°°°°°°°°°°°°°°°°°°°°°°°°°°°°°°°°°°°°°°°°°°°°°°°°°°°°
   //
   ELSIF #Sts.WorkModeMatCounter THEN


       // CASE 21 -> working mode = Material Counters; 100% when syncro running 
       // 
       IF #Sts.SynchroRunning AND NOT #Ctrl.Sync_EntryReduceOrStopFeed THEN
           #Ctrl.Entry_VelocityOverride := 100.0;
           #Sts.Cases_Entry_VelocityOverride := #ENTRY_CASE_21_V100_SYNCHRO_RUNNING;


       // CASE 22 -> working mode = Material Counters; 0% when syncro running  & work mode with STOP request 
       // 
       ELSIF #Sts.SynchroRunning AND #Ctrl.Sync_EntryReduceOrStopFeed AND (#PersistentValues.Par.SyncEntryMode = 1) THEN
           #Ctrl.Entry_VelocityOverride := 0.0;
           #Sts.Cases_Entry_VelocityOverride := #ENTRY_CASE_22_V0_SYNCHRO_RUNNING;


       // CASE 23 -> working mode = Material Counters; VMin when syncro running & work mode with REDUCE request
       // 
       ELSIF #Sts.SynchroRunning AND #Ctrl.Sync_EntryReduceOrStopFeed AND (#PersistentValues.Par.SyncEntryMode = 0) THEN
           #Ctrl.Entry_VelocityOverride := #PersistentValues.Par.Entry_Override1_VMin;
           #Sts.Cases_Entry_VelocityOverride := #ENTRY_CASE_23_VMin_SYNCHRO_RUNNING;


       // CASE 24 -> working mode = Material Counters; VMin if less then Limit 1 Position (material near to max loop position)
       // 
       ELSIF #Sts.LoopMaterialMissingToMaxLow < (#PersistentValues.Par.Entry_Lim1_VMin * #Sts.SelectedOverrideScaling) THEN
           #Ctrl.Entry_VelocityOverride := #PersistentValues.Par.Entry_Override1_VMin;
           #Sts.Cases_Entry_VelocityOverride := #ENTRY_CASE_24_VMin_MODE_COUNTERS;


       // CASE 25 -> working mode = Material Counters; VMed if less then Limit 2 Position (material in the middle loop position)
       // 
       ELSIF #Sts.LoopMaterialMissingToMaxLow < (#PersistentValues.Par.Entry_Lim2_VMed * #Sts.SelectedOverrideScaling) THEN
           #Ctrl.Entry_VelocityOverride := #PersistentValues.Par.Entry_Override2_VMed;
           #Sts.Cases_Entry_VelocityOverride := #ENTRY_CASE_25_VMed_MODE_COUNTERS;


       // CASE 26 -> working mode = Material Counters; VMax if less then Limit 3 Position (material far from the max loop position)
       // 
       ELSIF #Sts.LoopMaterialMissingToMaxLow < (#PersistentValues.Par.Entry_Lim3_VMax * #Sts.SelectedOverrideScaling) THEN
           #Ctrl.Entry_VelocityOverride := #PersistentValues.Par.Entry_Override3_VMax;
           #Sts.Cases_Entry_VelocityOverride := #ENTRY_CASE_26_VMax_MODE_COUNTERS;

       // CASE 27 -> working mode = Material Counters; VMax + 10% if greater then Limit 3 Position (material far from the max loop position)
       //     
       ELSE
           #Ctrl.Entry_VelocityOverride := MAX(IN1:=100.0,IN2:=(#PersistentValues.Par.Entry_Override3_VMax * 1.1));
           #Sts.Cases_Entry_VelocityOverride := #ENTRY_CASE_27_VMaxMax_MODE_COUNTERS;
       END_IF;


   // CASE 30 -> 100% if Unknown case
   // 
   ELSE
       #Ctrl.Entry_VelocityOverride := 100.0;
       #Sts.Cases_Entry_VelocityOverride := #ENTRY_CASE_30_V100_UNKNOW;
   END_IF;
END_REGION

REGION Network 41 (SCL): Exit machine velocity override
   // CASE 01 -> 0% when alarm presence
   // 
   IF #Sts.AlarmsPresence THEN

       #Ctrl.Exit_VelocityOverride := 0.0;
       #Sts.Cases_Exit_VelocityOverride := #EXIT_CASE_01_V0_ALARM_PRESENCE;


   // CASE 05 -> VMax when system is off and emptying confirmed
   // 
   ELSIF NOT #Sts.SystemOn
       AND
       (#CIn.Entry_EmptyingConfirmed
       OR
       ((NOT #DataIn.SensorEntryMaterialPresence OR #AreaInterfaceEntry.Man) AND NOT #DataIn.SensorExitMaterialPresence)
       )
   THEN
       #Ctrl.Exit_VelocityOverride := 100.0;
       #Sts.Cases_Exit_VelocityOverride := #EXIT_CASE_05_VMax_EMPTYING;


   // CASE 02 -> 0% when min high reached
   // 
   ELSIF #Sts.MinHighReached THEN
       #Ctrl.Exit_VelocityOverride := 0.0;
       #Sts.Cases_Exit_VelocityOverride := #EXIT_CASE_02_0_MIN_HIGH;



   // CASE 03 -> VMin when system is off
   // 
   ELSIF NOT #Sts.SystemOn AND NOT #CIn.Entry_EmptyingConfirmed THEN

       #Ctrl.Exit_VelocityOverride := #PersistentValues.Par.Exit_Override1_VMin;

       IF #AreaInterfaceExit.Man THEN
           #Ctrl.Exit_VelocityOverride := 100.0;
       END_IF;


       #Sts.Cases_Exit_VelocityOverride := #EXIT_CASE_03_VMin_SYSTEM_OFF;



   // CASE 04 -> VMin when entry next emptying 
   // 
   ELSIF #CIn.Entry_NxtEndOfMaterial THEN

       #Ctrl.Exit_VelocityOverride := #PersistentValues.Par.Exit_Override1_VMin;
       #Sts.Cases_Exit_VelocityOverride := #EXIT_CASE_04_VMin_NEXT_EMPTYING;



   //    
   //#################################################################################################################################
   // CASES When working mode = Sensors
   //#################################################################################################################################
   //
   ELSIF #Sts.WorkModeSensors THEN

       IF NOT (#PersistentValues.Par.WorkMode = #MODE_01_USE_MATERIAL_COUNTERS) OR #AreaInterfaceExit.Man THEN

           //CASE 11 -> working mode = Sensors; 100% if not the previous 
           #Ctrl.Exit_VelocityOverride := 100.0;
           #Sts.Cases_Exit_VelocityOverride := #EXIT_CASE_11_V100_MODE_SENSORS_OR_EXIT_MAN;
       ELSE
           //CASE 11 -> working mode = Sensors; 100% if not the previous 
           #Ctrl.Exit_VelocityOverride := #PersistentValues.Par.Exit_Override1_VMin;
           #Sts.Cases_Exit_VelocityOverride := #EXIT_CASE_12_VMIN_MODE_SENSORS_TEMPORARY;
       END_IF;




   //    
   //#################################################################################################################################
   // CASES  When working mode = Material Counters
   //#################################################################################################################################
   //

   ELSIF #Sts.WorkModeMatCounter THEN

       // CASE 20 -> working mode = Material Counters; 100% when syncro running and no reduce/stop request & work mode with stop request 
       // 
       IF #Sts.SynchroRunning AND NOT #Ctrl.Sync_ExitReduceOrStopFeed AND (#PersistentValues.Par.SyncExitMode = 1) THEN
           #Ctrl.Exit_VelocityOverride := 100.0;
           #Sts.Cases_Exit_VelocityOverride := #EXIT_CASE_20_100_SYNCRO_RUNNING;

       // CASE 21 -> working mode = Material Counters; 0% when syncro running & work mode with stop request 
       // 
       ELSIF #Sts.SynchroRunning AND #Ctrl.Sync_ExitReduceOrStopFeed AND (#PersistentValues.Par.SyncExitMode = 1) THEN
           #Ctrl.Exit_VelocityOverride := 0.0;
           #Sts.Cases_Exit_VelocityOverride := #EXIT_CASE_21_0_SYNCRO_RUNNING;


       // CASE 22 -> working mode = Material Counters; 100% when syncro running and work mode with reduce request
       // !!! RALLENTAMENTO GESTITO ESTERNAMENTE !!!
       ELSIF #Sts.SynchroRunning (*AND Ctrl.Sync_ExitReduceOrStopFeed*)AND (#PersistentValues.Par.SyncExitMode = 0) THEN
           #Ctrl.Exit_VelocityOverride := 100.0; // PersistentValue.Par.Exit_Override1_VMin; 
           #Sts.Cases_Exit_VelocityOverride := #EXIT_CASE_22_VMin_SYNCRO_RUNNING;



       // CASE 23 -> working mode = Material Counters; VMin IF less THEN Limit 1 Position (material near TO the min loop)
       // 
       ELSIF #Sts.LoopMaterialMissingToMinHigh <= #PersistentValues.Par.Exit_Lim1_VMin  THEN
           #Ctrl.Exit_VelocityOverride := #PersistentValues.Par.Exit_Override1_VMin;
           #Sts.Cases_Exit_VelocityOverride := #EXIT_CASE_23_VMin_MODE_COUNTERS;

       // CASE 24 -> working mode = Material Counters; VMed if less then Limit 2 Position (material in the middle loop position)
       // 
       ELSIF #Sts.LoopMaterialMissingToMinHigh <= #PersistentValues.Par.Exit_Lim2_VMed THEN
           #Ctrl.Exit_VelocityOverride := #PersistentValues.Par.Exit_Override2_VMed;
           #Sts.Cases_Exit_VelocityOverride := #EXIT_CASE_24_VMed_MODE_COUNTERS;

       // CASE 25 -> working mode = Material Counters; VMax if less then Limit 3 Position (material far from the min loop)
       // 
       ELSIF #Sts.LoopMaterialMissingToMinHigh <= #PersistentValues.Par.Exit_Lim3_VMax THEN
           #Ctrl.Exit_VelocityOverride := #PersistentValues.Par.Exit_Override3_VMax;
           #Sts.Cases_Exit_VelocityOverride := #EXIT_CASE_25_VMax_MODE_COUNTERS;

       // CASE 26 -> working mode = Material Counters; 100% if not the previous  
       // 
       ELSE
           #Ctrl.Exit_VelocityOverride := MAX_LREAL(IN1:=100.0,IN2:=#PersistentValues.Par.Exit_Override3_VMax);
           #Sts.Cases_Exit_VelocityOverride := #EXIT_CASE_26_100_MODE_COUNTERS;
       END_IF;

       // CASE 00 -> 0%
   ELSE
       #Ctrl.Exit_VelocityOverride := 0.0;
       #Sts.Cases_Exit_VelocityOverride := 0;
   END_IF;
END_REGION

REGION Network 42: Exit max allowable feeding
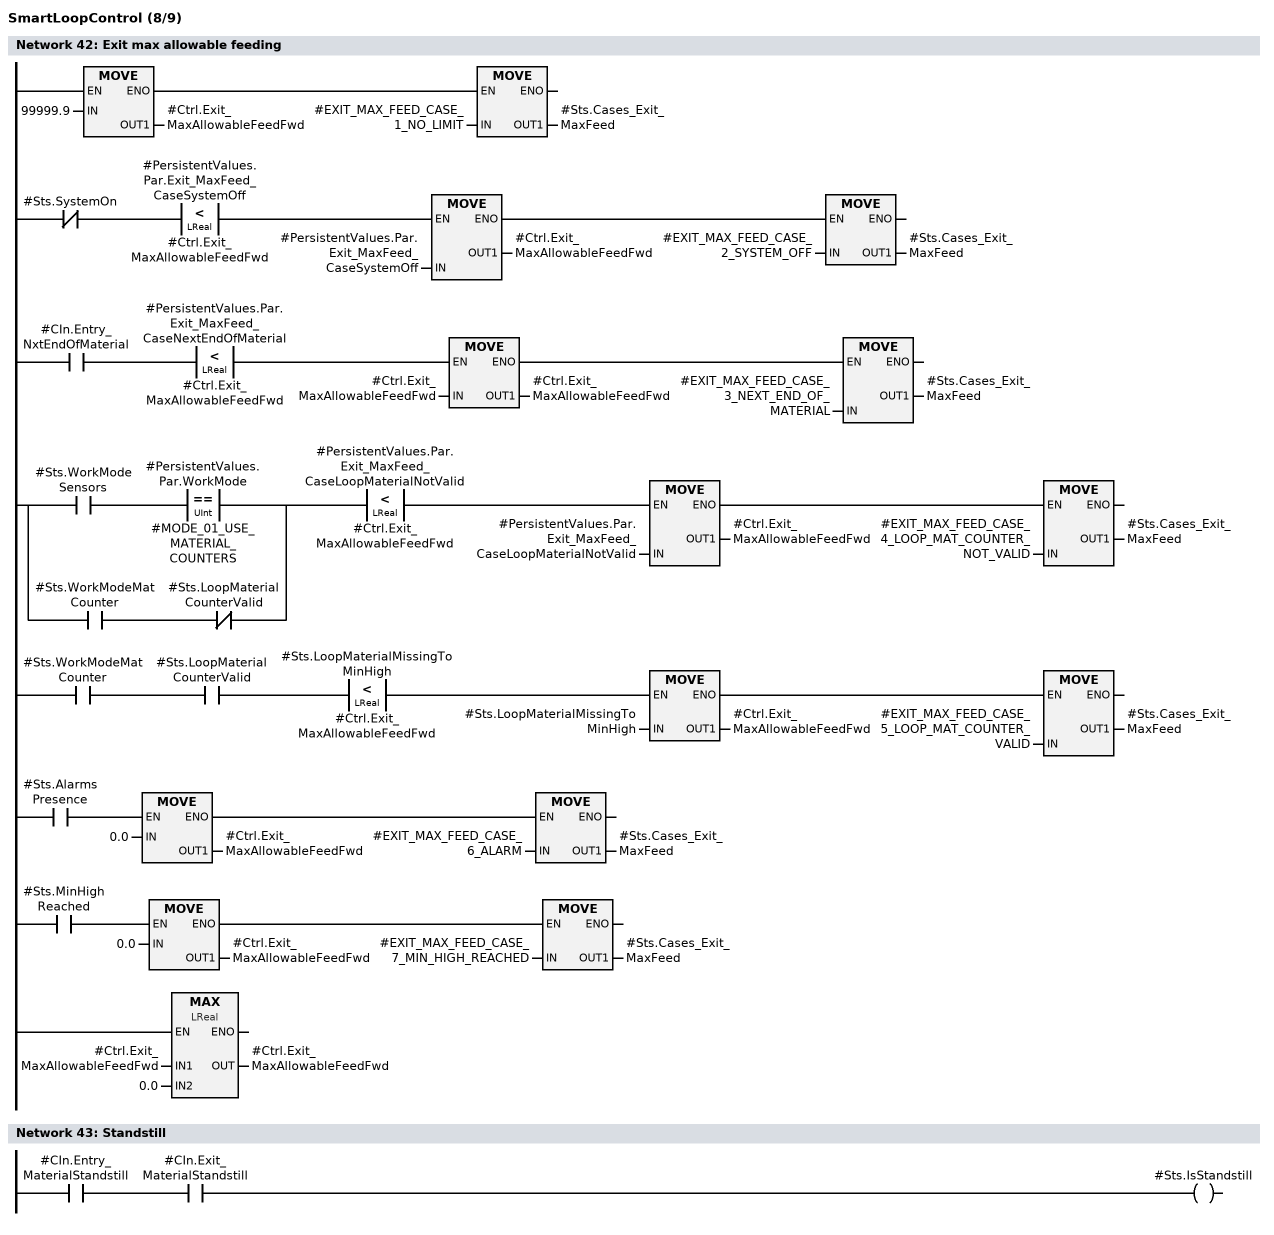
   RUNG wire#powerrail
      { S7_GenerateENO := "TRUE" } Move(in := 99999.9, out1 => #Ctrl.Exit_MaxAllowableFeedFwd)
      { S7_GenerateENO := "TRUE" } Move(in := #EXIT_MAX_FEED_CASE_1_NO_LIMIT, out1 => #Sts.Cases_Exit_MaxFeed)
   END_RUNG
   RUNG wire#powerrail
      I_Contact( #Sts.SystemOn )
      { S7_Templates := "SrcType := LReal" } LT_Contact(in1 := #PersistentValues.Par.Exit_MaxFeed_CaseSystemOff, in2 := #Ctrl.Exit_MaxAllowableFeedFwd)
      { S7_GenerateENO := "TRUE" } Move(in := #PersistentValues.Par.Exit_MaxFeed_CaseSystemOff, out1 => #Ctrl.Exit_MaxAllowableFeedFwd)
      { S7_GenerateENO := "TRUE" } Move(in := #EXIT_MAX_FEED_CASE_2_SYSTEM_OFF, out1 => #Sts.Cases_Exit_MaxFeed)
   END_RUNG
   RUNG wire#powerrail
      Contact( #CIn.Entry_NxtEndOfMaterial )
      { S7_Templates := "SrcType := LReal" } LT_Contact(in1 := #PersistentValues.Par.Exit_MaxFeed_CaseNextEndOfMaterial, in2 := #Ctrl.Exit_MaxAllowableFeedFwd)
      { S7_GenerateENO := "TRUE" } Move(in := #Ctrl.Exit_MaxAllowableFeedFwd, out1 => #Ctrl.Exit_MaxAllowableFeedFwd)
      { S7_GenerateENO := "TRUE" } Move(in := #EXIT_MAX_FEED_CASE_3_NEXT_END_OF_MATERIAL, out1 => #Sts.Cases_Exit_MaxFeed)
   END_RUNG
   RUNG wire#powerrail
      Contact( #Sts.WorkModeSensors )
      { S7_Templates := "SrcType := UInt" } EQ_Contact(in1 := #PersistentValues.Par.WorkMode, in2 := #MODE_01_USE_MATERIAL_COUNTERS)
      wire#w1
      { S7_Templates := "SrcType := LReal" } LT_Contact(in1 := #PersistentValues.Par.Exit_MaxFeed_CaseLoopMaterialNotValid, in2 := #Ctrl.Exit_MaxAllowableFeedFwd)
      { S7_GenerateENO := "TRUE" } Move(in := #PersistentValues.Par.Exit_MaxFeed_CaseLoopMaterialNotValid, out1 => #Ctrl.Exit_MaxAllowableFeedFwd)
      { S7_GenerateENO := "TRUE" } Move(in := #EXIT_MAX_FEED_CASE_4_LOOP_MAT_COUNTER_NOT_VALID, out1 => #Sts.Cases_Exit_MaxFeed)
   END_RUNG
   RUNG wire#powerrail
      Contact( #Sts.WorkModeMatCounter )
      I_Contact( #Sts.LoopMaterialCounterValid )
   END_RUNG wire#w1
   RUNG wire#powerrail
      Contact( #Sts.WorkModeMatCounter )
      Contact( #Sts.LoopMaterialCounterValid )
      { S7_Templates := "SrcType := LReal" } LT_Contact(in1 := #Sts.LoopMaterialMissingToMinHigh, in2 := #Ctrl.Exit_MaxAllowableFeedFwd)
      { S7_GenerateENO := "TRUE" } Move(in := #Sts.LoopMaterialMissingToMinHigh, out1 => #Ctrl.Exit_MaxAllowableFeedFwd)
      { S7_GenerateENO := "TRUE" } Move(in := #EXIT_MAX_FEED_CASE_5_LOOP_MAT_COUNTER_VALID, out1 => #Sts.Cases_Exit_MaxFeed)
   END_RUNG
   RUNG wire#powerrail
      Contact( #Sts.AlarmsPresence )
      { S7_GenerateENO := "TRUE" } Move(in := 0.0, out1 => #Ctrl.Exit_MaxAllowableFeedFwd)
      { S7_GenerateENO := "TRUE" } Move(in := #EXIT_MAX_FEED_CASE_6_ALARM, out1 => #Sts.Cases_Exit_MaxFeed)
   END_RUNG
   RUNG wire#powerrail
      Contact( #Sts.MinHighReached )
      { S7_GenerateENO := "TRUE" } Move(in := 0.0, out1 => #Ctrl.Exit_MaxAllowableFeedFwd)
      { S7_GenerateENO := "TRUE" } Move(in := #EXIT_MAX_FEED_CASE_7_MIN_HIGH_REACHED, out1 => #Sts.Cases_Exit_MaxFeed)
   END_RUNG
   RUNG wire#powerrail
      { S7_Templates := "[card := 2, value_type := LReal]" } MAX(in1 := #Ctrl.Exit_MaxAllowableFeedFwd, in2 := 0.0, out => #Ctrl.Exit_MaxAllowableFeedFwd)
   END_RUNG
   // the same network as SCL:
   // ENO of a box is taken as its EN; it also drops when the box reports an error
   #Ctrl.Exit_MaxAllowableFeedFwd := 99999.9;
   #Sts.Cases_Exit_MaxFeed := #EXIT_MAX_FEED_CASE_1_NO_LIMIT;
   #_w1 := NOT #Sts.SystemOn AND (#PersistentValues.Par.Exit_MaxFeed_CaseSystemOff < #Ctrl.Exit_MaxAllowableFeedFwd);
   IF #_w1 THEN
       #Ctrl.Exit_MaxAllowableFeedFwd := #PersistentValues.Par.Exit_MaxFeed_CaseSystemOff;
       #Sts.Cases_Exit_MaxFeed := #EXIT_MAX_FEED_CASE_2_SYSTEM_OFF;
   END_IF;
   #_w2 := #CIn.Entry_NxtEndOfMaterial AND (#PersistentValues.Par.Exit_MaxFeed_CaseNextEndOfMaterial < #Ctrl.Exit_MaxAllowableFeedFwd);
   IF #_w2 THEN
       #Ctrl.Exit_MaxAllowableFeedFwd := #Ctrl.Exit_MaxAllowableFeedFwd;
       #Sts.Cases_Exit_MaxFeed := #EXIT_MAX_FEED_CASE_3_NEXT_END_OF_MATERIAL;
   END_IF;
   #_w3 := ((#Sts.WorkModeSensors AND (#PersistentValues.Par.WorkMode = #MODE_01_USE_MATERIAL_COUNTERS)) OR (#Sts.WorkModeMatCounter AND NOT #Sts.LoopMaterialCounterValid)) AND (#PersistentValues.Par.Exit_MaxFeed_CaseLoopMaterialNotValid < #Ctrl.Exit_MaxAllowableFeedFwd);
   IF #_w3 THEN
       #Ctrl.Exit_MaxAllowableFeedFwd := #PersistentValues.Par.Exit_MaxFeed_CaseLoopMaterialNotValid;
       #Sts.Cases_Exit_MaxFeed := #EXIT_MAX_FEED_CASE_4_LOOP_MAT_COUNTER_NOT_VALID;
   END_IF;
   #_w4 := #Sts.WorkModeMatCounter AND #Sts.LoopMaterialCounterValid AND (#Sts.LoopMaterialMissingToMinHigh < #Ctrl.Exit_MaxAllowableFeedFwd);
   IF #_w4 THEN
       #Ctrl.Exit_MaxAllowableFeedFwd := #Sts.LoopMaterialMissingToMinHigh;
       #Sts.Cases_Exit_MaxFeed := #EXIT_MAX_FEED_CASE_5_LOOP_MAT_COUNTER_VALID;
   END_IF;
   IF #Sts.AlarmsPresence THEN
       #Ctrl.Exit_MaxAllowableFeedFwd := 0.0;
       #Sts.Cases_Exit_MaxFeed := #EXIT_MAX_FEED_CASE_6_ALARM;
   END_IF;
   IF #Sts.MinHighReached THEN
       #Ctrl.Exit_MaxAllowableFeedFwd := 0.0;
       #Sts.Cases_Exit_MaxFeed := #EXIT_MAX_FEED_CASE_7_MIN_HIGH_REACHED;
   END_IF;
   #Ctrl.Exit_MaxAllowableFeedFwd := MAX(IN1 := #Ctrl.Exit_MaxAllowableFeedFwd, IN2 := 0.0);
END_REGION

REGION Network 43: Standstill
   RUNG wire#powerrail
      Contact( #CIn.Entry_MaterialStandstill )
      Contact( #CIn.Exit_MaterialStandstill )
      Coil( #Sts.IsStandstill )
   END_RUNG
   // the same network as SCL:
   #Sts.IsStandstill := #CIn.Entry_MaterialStandstill AND #CIn.Exit_MaterialStandstill;
END_REGION

REGION Network 44: Alarms presence
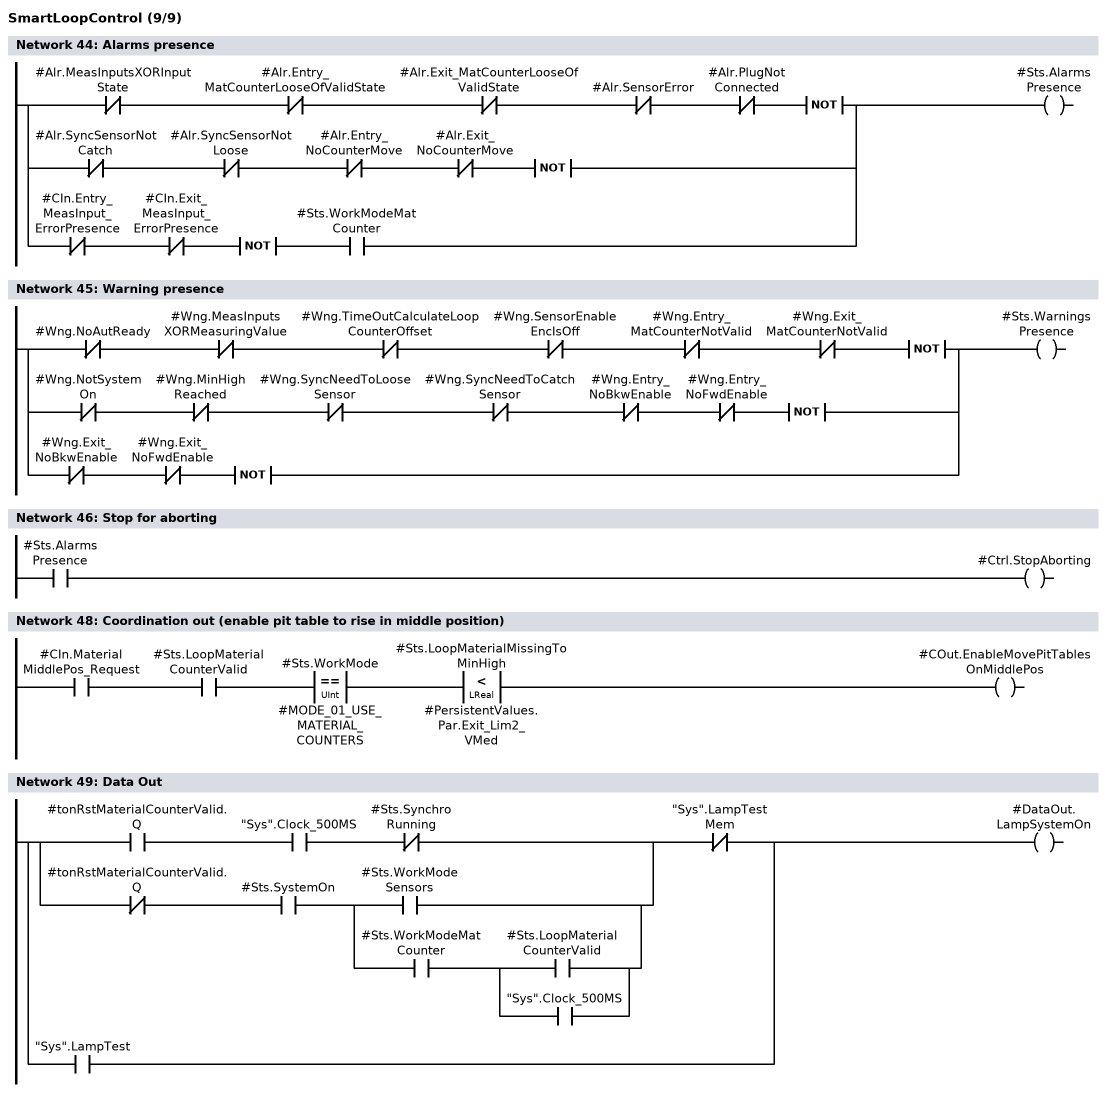
   RUNG wire#powerrail
      I_Contact( #Alr.MeasInputsXORInputState )
      I_Contact( #Alr.Entry_MatCounterLooseOfValidState )
      I_Contact( #Alr.Exit_MatCounterLooseOfValidState )
      I_Contact( #Alr.SensorError )
      I_Contact( #Alr.PlugNotConnected )
      Not()
      wire#w1
      Coil( #Sts.AlarmsPresence )
   END_RUNG
   RUNG wire#powerrail
      I_Contact( #Alr.SyncSensorNotCatch )
      I_Contact( #Alr.SyncSensorNotLoose )
      I_Contact( #Alr.Entry_NoCounterMove )
      I_Contact( #Alr.Exit_NoCounterMove )
      Not()
   END_RUNG wire#w1
   RUNG wire#powerrail
      I_Contact( #CIn.Entry_MeasInput_ErrorPresence )
      I_Contact( #CIn.Exit_MeasInput_ErrorPresence )
      Not()
      Contact( #Sts.WorkModeMatCounter )
   END_RUNG wire#w1
   // the same network as SCL:
   #Sts.AlarmsPresence := NOT (NOT #Alr.MeasInputsXORInputState AND NOT #Alr.Entry_MatCounterLooseOfValidState AND NOT #Alr.Exit_MatCounterLooseOfValidState AND NOT #Alr.SensorError AND NOT #Alr.PlugNotConnected) OR NOT (NOT #Alr.SyncSensorNotCatch AND NOT #Alr.SyncSensorNotLoose AND NOT #Alr.Entry_NoCounterMove AND NOT #Alr.Exit_NoCounterMove) OR (NOT (NOT #CIn.Entry_MeasInput_ErrorPresence AND NOT #CIn.Exit_MeasInput_ErrorPresence) AND #Sts.WorkModeMatCounter);
END_REGION

REGION Network 45: Warning presence
   RUNG wire#powerrail
      I_Contact( #Wng.NoAutReady )
      I_Contact( #Wng.MeasInputsXORMeasuringValue )
      I_Contact( #Wng.TimeOutCalculateLoopCounterOffset )
      I_Contact( #Wng.SensorEnableEncIsOff )
      I_Contact( #Wng.Entry_MatCounterNotValid )
      I_Contact( #Wng.Exit_MatCounterNotValid )
      Not()
      wire#w1
      Coil( #Sts.WarningsPresence )
   END_RUNG
   RUNG wire#powerrail
      I_Contact( #Wng.NotSystemOn )
      I_Contact( #Wng.MinHighReached )
      I_Contact( #Wng.SyncNeedToLooseSensor )
      I_Contact( #Wng.SyncNeedToCatchSensor )
      I_Contact( #Wng.Entry_NoBkwEnable )
      I_Contact( #Wng.Entry_NoFwdEnable )
      Not()
   END_RUNG wire#w1
   RUNG wire#powerrail
      I_Contact( #Wng.Exit_NoBkwEnable )
      I_Contact( #Wng.Exit_NoFwdEnable )
      Not()
   END_RUNG wire#w1
   // the same network as SCL:
   #Sts.WarningsPresence := NOT (NOT #Wng.NoAutReady AND NOT #Wng.MeasInputsXORMeasuringValue AND NOT #Wng.TimeOutCalculateLoopCounterOffset AND NOT #Wng.SensorEnableEncIsOff AND NOT #Wng.Entry_MatCounterNotValid AND NOT #Wng.Exit_MatCounterNotValid) OR NOT (NOT #Wng.NotSystemOn AND NOT #Wng.MinHighReached AND NOT #Wng.SyncNeedToLooseSensor AND NOT #Wng.SyncNeedToCatchSensor AND NOT #Wng.Entry_NoBkwEnable AND NOT #Wng.Entry_NoFwdEnable) OR NOT (NOT #Wng.Exit_NoBkwEnable AND NOT #Wng.Exit_NoFwdEnable);
END_REGION

REGION Network 46: Stop for aborting
   RUNG wire#powerrail
      Contact( #Sts.AlarmsPresence )
      Coil( #Ctrl.StopAborting )
   END_RUNG
   // the same network as SCL:
   #Ctrl.StopAborting := #Sts.AlarmsPresence;
END_REGION

REGION Network 47 (SCL): Coordination out
   #COut.SystemOn := #Sts.SystemOn;
   #COut.LoopMaterialCounterValid := #Sts.LoopMaterialCounterValid;
   #COut.MaxLowReached := #Sts.MaxLowReached;
   #COut.MinHighReached := #Sts.MinHighReached;
   #COut.SynchroRunning := #Sts.SynchroRunning;
   #COut.SynchroDone := #Sts.SynchroDoneTof2s;
   #COut.Sync_EntryReduceOrStopFeed := #Ctrl.Sync_EntryReduceOrStopFeed;
   #COut.Sync_ExitReduceOrStopFeed := #Ctrl.Sync_ExitReduceOrStopFeed;
   #COut.Entry_EnableFeedBkw := #Ctrl.Entry_EnableFeedBkw;
   #COut.Entry_EnableFeedFwd := #Ctrl.Entry_EnableFeedFwd;
   #COut.Exit_EnableFeedBkw := #Ctrl.Exit_EnableFeedBkw;
   #COut.Exit_EnableFeedFwd := #Ctrl.Exit_EnableFeedFwd;
   #COut.EnableMeasuringInputs := #Ctrl.MeasuringEnable;

   #COut.LoopMaterialCounter := #Sts.LoopMaterialCounter;
   #COut.LoopMaterialMissingToSynch := #Sts.MissingToCyclicSync;
   #COut.LoopMaterialMissingToMaxLow := #Sts.LoopMaterialMissingToMaxLow;
   #COut.LoopMaterialMissingToMinHigh := #Sts.LoopMaterialMissingToMinHigh;
   #COut.Entry_ActVelocityOverride := #Sts.Cases_Entry_VelocityOverride;
   #COut.Exit_ActVelocityOverride := #Sts.Cases_Exit_VelocityOverride;
   #COut.Entry_VelocityOverride := #Ctrl.Entry_VelocityOverride;
   #COut.Exit_VelocityOverride := #Ctrl.Exit_VelocityOverride;
   #COut.Exit_MaxAllowableFeedFwd := #Ctrl.Exit_MaxAllowableFeedFwd;
END_REGION

REGION Network 48: Coordination out (enable pit table to rise in middle position)
   RUNG wire#powerrail
      Contact( #CIn.MaterialMiddlePos_Request )
      Contact( #Sts.LoopMaterialCounterValid )
      { S7_Templates := "SrcType := UInt" } EQ_Contact(in1 := #Sts.WorkMode, in2 := #MODE_01_USE_MATERIAL_COUNTERS)
      { S7_Templates := "SrcType := LReal" } LT_Contact(in1 := #Sts.LoopMaterialMissingToMinHigh, in2 := #PersistentValues.Par.Exit_Lim2_VMed)
      Coil( #COut.EnableMovePitTablesOnMiddlePos )
   END_RUNG
   // the same network as SCL:
   #COut.EnableMovePitTablesOnMiddlePos := #CIn.MaterialMiddlePos_Request AND #Sts.LoopMaterialCounterValid AND (#Sts.WorkMode = #MODE_01_USE_MATERIAL_COUNTERS) AND (#Sts.LoopMaterialMissingToMinHigh < #PersistentValues.Par.Exit_Lim2_VMed);
END_REGION

REGION Network 49: Data Out
   RUNG wire#powerrail
      Contact( #tonRstMaterialCounterValid.Q )
      Contact( "Sys".Clock_500MS )
      I_Contact( #Sts.SynchroRunning )
      wire#w1
      I_Contact( "Sys".LampTestMem )
      wire#w4
      Coil( #DataOut.LampSystemOn )
   END_RUNG
   RUNG wire#powerrail
      I_Contact( #tonRstMaterialCounterValid.Q )
      Contact( #Sts.SystemOn )
      wire#w2
      Contact( #Sts.WorkModeSensors )
   END_RUNG wire#w1
   RUNG wire#w2
      Contact( #Sts.WorkModeMatCounter )
      wire#w3
      Contact( #Sts.LoopMaterialCounterValid )
   END_RUNG wire#w1
   RUNG wire#w3
      Contact( "Sys".Clock_500MS )
   END_RUNG wire#w1
   RUNG wire#powerrail
      Contact( "Sys".LampTest )
   END_RUNG wire#w4
   // the same network as SCL:
   #DataOut.LampSystemOn := (((#tonRstMaterialCounterValid.Q AND "Sys".Clock_500MS AND NOT #Sts.SynchroRunning) OR (NOT #tonRstMaterialCounterValid.Q AND #Sts.SystemOn AND (#Sts.WorkModeSensors OR (#Sts.WorkModeMatCounter AND (#Sts.LoopMaterialCounterValid OR "Sys".Clock_500MS))))) AND NOT "Sys".LampTestMem) OR "Sys".LampTest;
END_REGION

REGION Network 50 (SCL): Entry machine interface
   // Status machine ready
   #MachineInterfaceEntry.AutReady := #AreaInterfaceEntry.Aut AND NOT #Sts.AlarmsPresence;
   // Status machine aborting
   #MachineInterfaceEntry.Aborting := #Ctrl.StopAborting;
   // Status Ack Stop in phase
   #MachineInterfaceEntry.AckStopInPhase := #Ctrl.StopInPhase AND #MachineInterfaceEntry.MotionsStandStill;
   // Status Ack Stop programmed
   #MachineInterfaceEntry.AckStopProgrammed := #Ctrl.StopProgrammed AND #MachineInterfaceEntry.MotionsStandStill;
   // Status Motion standtill
   #MachineInterfaceEntry.MotionsStandStill := #Sts.IsStandstill;
   // Status Alarm presence
   #MachineInterfaceEntry.AlarmsPresence := #Sts.AlarmsPresence;
   // Status Warning presence
   #MachineInterfaceEntry.WarningPresence := #Sts.WarningsPresence;


   // Warning machine not automatic ready
   IF #AreaInterfaceEntry.CheckAutReady AND NOT #MachineInterfaceEntry.AutReady THEN
       #Wng.NoAutReady := TRUE;
   END_IF;
END_REGION

REGION Network 51 (SCL): Exit machine interface
   // Status machine ready
   #MachineInterfaceExit.AutReady := #AreaInterfaceExit.Aut AND NOT #Sts.AlarmsPresence;
   // Status machine auto
   // Status machine aborting
   #MachineInterfaceExit.Aborting := #Ctrl.StopAborting;
   // Status Ack Stop in phase
   #MachineInterfaceExit.AckStopInPhase := #Ctrl.StopInPhase AND #MachineInterfaceExit.MotionsStandStill;
   // Status Ack Stop programmed
   #MachineInterfaceExit.AckStopProgrammed := #Ctrl.StopProgrammed AND #MachineInterfaceExit.MotionsStandStill;
   // Status Motion standtill
   #MachineInterfaceExit.MotionsStandStill := #Sts.IsStandstill;
   // Status Alarm presence
   #MachineInterfaceExit.AlarmsPresence := #Sts.AlarmsPresence;
   // Status Warning presence
   #MachineInterfaceExit.WarningPresence := #Sts.WarningsPresence;


   // Warning machine not automatic ready
   IF #AreaInterfaceExit.CheckAutReady AND NOT #MachineInterfaceExit.AutReady THEN
       #Wng.NoAutReady := TRUE;
   END_IF;
END_REGION
END_FUNCTION_BLOCK
